Universal Robots PolyScope program: set_b_drawing_robot.urp

Program set_b_drawing_robot (installation=default directory=/programs createdIn=5.11.9.1010452 lastSavedIn=5.11.9.1010452 robotSerialNumber=20225200364)
Calibrated DH parameters: a=[0.00002, -0.569483, -0.54992, -0.00001, -0.000036, 0]; d=[0.180894, -146.691669, 192.918669, -46.053088, 0.119778, 0.115602]; alpha=[1.571425, -0.001534, 0.003359, 1.568739, -1.571477, 0]; deltaTheta=[0, 0.376258, -0.101074, -0.275185, -0.000002, 0]
Robot Program (runOnlyOnce=true)
  Script file /programs/set_b_drawing_robot.script_bak
    | def Machining3():
    |   # Default parameters:
    |   global speed_ms = 0.3
    |   global speed_rads = 0.75
    |   global accel_mss = 3
    |   global accel_radss = 1.2
    |   global blend_radius_m = 0.00001
    | 
    |   # Add subprograms here
    |   # Start of main program
    |   # Program generated by RoboDK v5.6.5 for UR10e on 17/10/2023 11:45:54
    |   # Using nominal kinematics.
    |   blend_radius_m = 0.001
    |   speed_ms = 1.000
    |   # set_reference(p[0.335000, -0.154000, -0.015000, 0.000000, 0.000000, 0.000000])
    |   set_tcp(p[0.000000, 0.000000, 0.252000, 0.000000, 0.000000, 0.000000])
    |   # Show Tool
    |   movej([0.061043, -1.072595, -2.581751, -1.058043, 1.570796, 1.631840],accel_radss,speed_rads,0,blend_radius_m)
    |   movel([0.061043, -1.163101, -2.647930, -0.901358, 1.570796, 1.631840],accel_mss,speed_ms,0,blend_radius_m)
    |   speed_ms = 1.000
    |   speed_ms = 0.005
    |   movel([0.061043, -1.123091, -2.622268, -0.967030, 1.570796, 1.631840],accel_mss,speed_ms,0,blend_radius_m)
    |   speed_ms = 1.000
    |   movel([0.061043, -1.163101, -2.647930, -0.901358, 1.570796, 1.631840],accel_mss,speed_ms,0,blend_radius_m)
    |   speed_ms = 0.040
    |   speed_ms = 1.000
    |   movel([0.083343, -1.403315, -2.504510, -0.804564, 1.570796, 1.654139],accel_mss,speed_ms,0,blend_radius_m)
    |   speed_ms = 0.005
    |   movel([0.083343, -1.443044, -2.523768, -0.745577, 1.570796, 1.654139],accel_mss,speed_ms,0,blend_radius_m)
    |   speed_ms = 0.035
    |   movel([0.081487, -1.443536, -2.523375, -0.745478, 1.570796, 1.652283],accel_mss,speed_ms,0,blend_radius_m)
    |   movel([0.082098, -1.437213, -2.528399, -0.746777, 1.570796, 1.652894],accel_mss,speed_ms,0,blend_radius_m)
    |   movel([0.082718, -1.430832, -2.533407, -0.748150, 1.570796, 1.653514],accel_mss,speed_ms,0,blend_radius_m)
    |   movel([0.084603, -1.430324, -2.533803, -0.748261, 1.570796, 1.655399],accel_mss,speed_ms,0,blend_radius_m)
    |   movel([0.086489, -1.429818, -2.534197, -0.748373, 1.570796, 1.657285],accel_mss,speed_ms,0,blend_radius_m)
    |   movel([0.085840, -1.436215, -2.529186, -0.746988, 1.570796, 1.656636],accel_mss,speed_ms,0,blend_radius_m)
    |   movel([0.085200, -1.442554, -2.524159, -0.745676, 1.570796, 1.655996],accel_mss,speed_ms,0,blend_radius_m)
    |   movel([0.083343, -1.443044, -2.523768, -0.745577, 1.570796, 1.654139],accel_mss,speed_ms,0,blend_radius_m)
    |   movel([0.081487, -1.443536, -2.523375, -0.745478, 1.570796, 1.652283],accel_mss,speed_ms,0,blend_radius_m)
    |   movel([0.081525, -1.443142, -2.523689, -0.745557, 1.570796, 1.652321],accel_mss,speed_ms,0,blend_radius_m)
    |   speed_ms = 0.005
    |   movel([0.081525, -1.434929, -2.519954, -0.757506, 1.570796, 1.652321],accel_mss,speed_ms,0,blend_radius_m)
    |   speed_ms = 0.040
    |   movel([0.115333, -1.443644, -2.513024, -0.755721, 1.570796, 1.686129],accel_mss,speed_ms,0,blend_radius_m)
    |   speed_ms = 0.005
    |   movel([0.115333, -1.451791, -2.516723, -0.743874, 1.570796, 1.686129],accel_mss,speed_ms,0,blend_radius_m)
    |   speed_ms = 0.035
    |   movel([0.102885, -1.454661, -2.514387, -0.743341, 1.570796, 1.673681],accel_mss,speed_ms,0,blend_radius_m)
    |   movel([0.102970, -1.452841, -2.515871, -0.743678, 1.570796, 1.673766],accel_mss,speed_ms,0,blend_radius_m)
    |   movel([0.103055, -1.451016, -2.517353, -0.744021, 1.570796, 1.673851],accel_mss,speed_ms,0,blend_radius_m)
    |   movel([0.115713, -1.447978, -2.519809, -0.744602, 1.570796, 1.686509],accel_mss,speed_ms,0,blend_radius_m)
    |   movel([0.128398, -1.445051, -2.522162, -0.745176, 1.570796, 1.699194],accel_mss,speed_ms,0,blend_radius_m)
    |   movel([0.128100, -1.447044, -2.520561, -0.744784, 1.570796, 1.698897],accel_mss,speed_ms,0,blend_radius_m)
    |   movel([0.127804, -1.449031, -2.518959, -0.744399, 1.570796, 1.698600],accel_mss,speed_ms,0,blend_radius_m)
    |   movel([0.115333, -1.451791, -2.516723, -0.743874, 1.570796, 1.686129],accel_mss,speed_ms,0,blend_radius_m)
    |   movel([0.113047, -1.452309, -2.516303, -0.743777, 1.570796, 1.683843],accel_mss,speed_ms,0,blend_radius_m)
    |   speed_ms = 0.005
    |   movel([0.113047, -1.444166, -2.512605, -0.755618, 1.570796, 1.683843],accel_mss,speed_ms,0,blend_radius_m)
    |   speed_ms = 0.040
    |   movel([0.116068, -1.438174, -2.517387, -0.756828, 1.570796, 1.686864],accel_mss,speed_ms,0,blend_radius_m)
    |   speed_ms = 0.005
    |   movel([0.116068, -1.446363, -2.521109, -0.744917, 1.570796, 1.686864],accel_mss,speed_ms,0,blend_radius_m)
    |   speed_ms = 0.035
    |   movel([0.086775, -1.453581, -2.515268, -0.743540, 1.570796, 1.657571],accel_mss,speed_ms,0,blend_radius_m)
    |   movel([0.089171, -1.430471, -2.533689, -0.748229, 1.570796, 1.659968],accel_mss,speed_ms,0,blend_radius_m)
    |   movel([0.091706, -1.406568, -2.551895, -0.753926, 1.570796, 1.662503],accel_mss,speed_ms,0,blend_radius_m)
    |   movel([0.122816, -1.398387, -2.557932, -0.756070, 1.570796, 1.693612],accel_mss,speed_ms,0,blend_radius_m)
    |   movel([0.154099, -1.390862, -2.563398, -0.758129, 1.570796, 1.724895],accel_mss,speed_ms,0,blend_radius_m)
    |   movel([0.149681, -1.415746, -2.545005, -0.751638, 1.570796, 1.720477],accel_mss,speed_ms,0,blend_radius_m)
    |   movel([0.145508, -1.439740, -2.526398, -0.746251, 1.570796, 1.716304],accel_mss,speed_ms,0,blend_radius_m)
    |   movel([0.116068, -1.446363, -2.521109, -0.744917, 1.570796, 1.686864],accel_mss,speed_ms,0,blend_radius_m)
    |   movel([0.113764, -1.446908, -2.520670, -0.744811, 1.570796, 1.684560],accel_mss,speed_ms,0,blend_radius_m)
    |   speed_ms = 0.005
    |   movel([0.113764, -1.438723, -2.516951, -0.756715, 1.570796, 1.684560],accel_mss,speed_ms,0,blend_radius_m)
    |   speed_ms = 0.040
    |   movel([0.108373, -1.429267, -2.524395, -0.758727, 1.570796, 1.679169],accel_mss,speed_ms,0,blend_radius_m)
    |   speed_ms = 0.005
    |   movel([0.108373, -1.437523, -2.528153, -0.746712, 1.570796, 1.679169],accel_mss,speed_ms,0,blend_radius_m)
    |   speed_ms = 0.035
    |   movel([0.107038, -1.438547, -2.527344, -0.746498, 1.570796, 1.677835],accel_mss,speed_ms,0,blend_radius_m)
    |   movel([0.106310, -1.438957, -2.527019, -0.746413, 1.570796, 1.677107],accel_mss,speed_ms,0,blend_radius_m)
    |   movel([0.104799, -1.439542, -2.526555, -0.746292, 1.570796, 1.675596],accel_mss,speed_ms,0,blend_radius_m)
    |   movel([0.104044, -1.439704, -2.526426, -0.746258, 1.570796, 1.674840],accel_mss,speed_ms,0,blend_radius_m)
    |   movel([0.102614, -1.439758, -2.526384, -0.746247, 1.570796, 1.673411],accel_mss,speed_ms,0,blend_radius_m)
    |   movel([0.101980, -1.439648, -2.526471, -0.746270, 1.570796, 1.672776],accel_mss,speed_ms,0,blend_radius_m)
    |   movel([0.100905, -1.439161, -2.526857, -0.746371, 1.570796, 1.671701],accel_mss,speed_ms,0,blend_radius_m)
    |   movel([0.100487, -1.438793, -2.527149, -0.746447, 1.570796, 1.671284],accel_mss,speed_ms,0,blend_radius_m)
    |   movel([0.099966, -1.437859, -2.527888, -0.746642, 1.570796, 1.670762],accel_mss,speed_ms,0,blend_radius_m)
    |   movel([0.099866, -1.437301, -2.528329, -0.746759, 1.570796, 1.670663],accel_mss,speed_ms,0,blend_radius_m)
    |   movel([0.099878, -1.436700, -2.528804, -0.746885, 1.570796, 1.670674],accel_mss,speed_ms,0,blend_radius_m)
    |   movel([0.100054, -1.435839, -2.529482, -0.747068, 1.570796, 1.670850],accel_mss,speed_ms,0,blend_radius_m)
    |   movel([0.100376, -1.435105, -2.530060, -0.747224, 1.570796, 1.671172],accel_mss,speed_ms,0,blend_radius_m)
    |   movel([0.100937, -1.434333, -2.530667, -0.747389, 1.570796, 1.671733],accel_mss,speed_ms,0,blend_radius_m)
    |   movel([0.101867, -1.433331, -2.531453, -0.747605, 1.570796, 1.672664],accel_mss,speed_ms,0,blend_radius_m)
    |   movel([0.103005, -1.432248, -2.532301, -0.747840, 1.570796, 1.673801],accel_mss,speed_ms,0,blend_radius_m)
    |   movel([0.103766, -1.431710, -2.532722, -0.747957, 1.570796, 1.674563],accel_mss,speed_ms,0,blend_radius_m)
    |   movel([0.104600, -1.431387, -2.532974, -0.748028, 1.570796, 1.675397],accel_mss,speed_ms,0,blend_radius_m)
    |   movel([0.106011, -1.431098, -2.533199, -0.748091, 1.570796, 1.676807],accel_mss,speed_ms,0,blend_radius_m)
    |   movel([0.107167, -1.430973, -2.533297, -0.748119, 1.570796, 1.677964],accel_mss,speed_ms,0,blend_radius_m)
    |   movel([0.108266, -1.430998, -2.533278, -0.748113, 1.570796, 1.679062],accel_mss,speed_ms,0,blend_radius_m)
    |   movel([0.109099, -1.431186, -2.533131, -0.748072, 1.570796, 1.679896],accel_mss,speed_ms,0,blend_radius_m)
    |   movel([0.109775, -1.431571, -2.532831, -0.747988, 1.570796, 1.680572],accel_mss,speed_ms,0,blend_radius_m)
    |   movel([0.110228, -1.432115, -2.532405, -0.747869, 1.570796, 1.681024],accel_mss,speed_ms,0,blend_radius_m)
    |   movel([0.110459, -1.432805, -2.531865, -0.747719, 1.570796, 1.681255],accel_mss,speed_ms,0,blend_radius_m)
    |   movel([0.110489, -1.433683, -2.531177, -0.747529, 1.570796, 1.681285],accel_mss,speed_ms,0,blend_radius_m)
    |   movel([0.110328, -1.434616, -2.530445, -0.747328, 1.570796, 1.681124],accel_mss,speed_ms,0,blend_radius_m)
    |   movel([0.110059, -1.435334, -2.529880, -0.747175, 1.570796, 1.680855],accel_mss,speed_ms,0,blend_radius_m)
    |   movel([0.109634, -1.436071, -2.529299, -0.747018, 1.570796, 1.680430],accel_mss,speed_ms,0,blend_radius_m)
    |   movel([0.109064, -1.436811, -2.528716, -0.746862, 1.570796, 1.679861],accel_mss,speed_ms,0,blend_radius_m)
    |   movel([0.108373, -1.437523, -2.528153, -0.746712, 1.570796, 1.679169],accel_mss,speed_ms,0,blend_radius_m)
    |   movel([0.107038, -1.438547, -2.527344, -0.746498, 1.570796, 1.677835],accel_mss,speed_ms,0,blend_radius_m)
    |   movel([0.106310, -1.438957, -2.527019, -0.746413, 1.570796, 1.677107],accel_mss,speed_ms,0,blend_radius_m)
    |   speed_ms = 0.005
    |   movel([0.106310, -1.430712, -2.523266, -0.758411, 1.570796, 1.677107],accel_mss,speed_ms,0,blend_radius_m)
    |   speed_ms = 0.040
    |   movel([0.108450, -1.424967, -2.527736, -0.759686, 1.570796, 1.679246],accel_mss,speed_ms,0,blend_radius_m)
    |   speed_ms = 0.005
    |   movel([0.108450, -1.433255, -2.531513, -0.747621, 1.570796, 1.679246],accel_mss,speed_ms,0,blend_radius_m)
    |   speed_ms = 0.035
    |   movel([0.108678, -1.434176, -2.530790, -0.747423, 1.570796, 1.679474],accel_mss,speed_ms,0,blend_radius_m)
    |   movel([0.108589, -1.434982, -2.530157, -0.747250, 1.570796, 1.679385],accel_mss,speed_ms,0,blend_radius_m)
    |   movel([0.108163, -1.435793, -2.529519, -0.747077, 1.570796, 1.678959],accel_mss,speed_ms,0,blend_radius_m)
    |   movel([0.107355, -1.436726, -2.528783, -0.746880, 1.570796, 1.678151],accel_mss,speed_ms,0,blend_radius_m)
    |   movel([0.106463, -1.437462, -2.528202, -0.746725, 1.570796, 1.677259],accel_mss,speed_ms,0,blend_radius_m)
    |   movel([0.105461, -1.438014, -2.527765, -0.746609, 1.570796, 1.676258],accel_mss,speed_ms,0,blend_radius_m)
    |   movel([0.104454, -1.438323, -2.527521, -0.746545, 1.570796, 1.675251],accel_mss,speed_ms,0,blend_radius_m)
    |   movel([0.103505, -1.438364, -2.527489, -0.746536, 1.570796, 1.674302],accel_mss,speed_ms,0,blend_radius_m)
    |   movel([0.102703, -1.438137, -2.527668, -0.746584, 1.570796, 1.673500],accel_mss,speed_ms,0,blend_radius_m)
    |   movel([0.102119, -1.437659, -2.528047, -0.746684, 1.570796, 1.672915],accel_mss,speed_ms,0,blend_radius_m)
    |   movel([0.101790, -1.436965, -2.528595, -0.746830, 1.570796, 1.672586],accel_mss,speed_ms,0,blend_radius_m)
    |   movel([0.101749, -1.436130, -2.529253, -0.747006, 1.570796, 1.672545],accel_mss,speed_ms,0,blend_radius_m)
    |   movel([0.101858, -1.435631, -2.529646, -0.747112, 1.570796, 1.672655],accel_mss,speed_ms,0,blend_radius_m)
    |   movel([0.102363, -1.434622, -2.530440, -0.747327, 1.570796, 1.673159],accel_mss,speed_ms,0,blend_radius_m)
    |   movel([0.102745, -1.434142, -2.530817, -0.747430, 1.570796, 1.673541],accel_mss,speed_ms,0,blend_radius_m)
    |   movel([0.103728, -1.433264, -2.531506, -0.747619, 1.570796, 1.674524],accel_mss,speed_ms,0,blend_radius_m)
    |   movel([0.104871, -1.432616, -2.532013, -0.747760, 1.570796, 1.675667],accel_mss,speed_ms,0,blend_radius_m)
    |   movel([0.106038, -1.432273, -2.532282, -0.747834, 1.570796, 1.676835],accel_mss,speed_ms,0,blend_radius_m)
    |   movel([0.107121, -1.432265, -2.532288, -0.747836, 1.570796, 1.677918],accel_mss,speed_ms,0,blend_radius_m)
    |   movel([0.107572, -1.432389, -2.532191, -0.747809, 1.570796, 1.678368],accel_mss,speed_ms,0,blend_radius_m)
    |   movel([0.107952, -1.432601, -2.532025, -0.747763, 1.570796, 1.678748],accel_mss,speed_ms,0,blend_radius_m)
    |   movel([0.108450, -1.433255, -2.531513, -0.747621, 1.570796, 1.679246],accel_mss,speed_ms,0,blend_radius_m)
    |   movel([0.108678, -1.434176, -2.530790, -0.747423, 1.570796, 1.679474],accel_mss,speed_ms,0,blend_radius_m)
    |   movel([0.108589, -1.434982, -2.530157, -0.747250, 1.570796, 1.679385],accel_mss,speed_ms,0,blend_radius_m)
    |   speed_ms = 0.005
    |   movel([0.108509, -1.426858, -2.526270, -0.759261, 1.570796, 1.679305],accel_mss,speed_ms,0,blend_radius_m)
    |   speed_ms = 0.040
    |   movel([0.111498, -1.422635, -2.529536, -0.760218, 1.570796, 1.682294],accel_mss,speed_ms,0,blend_radius_m)
    |   speed_ms = 0.005
    |   movel([0.111498, -1.430940, -2.533323, -0.748126, 1.570796, 1.682294],accel_mss,speed_ms,0,blend_radius_m)
    |   speed_ms = 0.035
    |   movel([0.111769, -1.431458, -2.532919, -0.748012, 1.570796, 1.682566],accel_mss,speed_ms,0,blend_radius_m)
    |   movel([0.112066, -1.432871, -2.531814, -0.747704, 1.570796, 1.682862],accel_mss,speed_ms,0,blend_radius_m)
    |   movel([0.112043, -1.433534, -2.531294, -0.747561, 1.570796, 1.682839],accel_mss,speed_ms,0,blend_radius_m)
    |   movel([0.111849, -1.434440, -2.530583, -0.747366, 1.570796, 1.682646],accel_mss,speed_ms,0,blend_radius_m)
    |   movel([0.111503, -1.435363, -2.529857, -0.747169, 1.570796, 1.682299],accel_mss,speed_ms,0,blend_radius_m)
    |   movel([0.111013, -1.436281, -2.529134, -0.746974, 1.570796, 1.681809],accel_mss,speed_ms,0,blend_radius_m)
    |   movel([0.110389, -1.437172, -2.528431, -0.746786, 1.570796, 1.681185],accel_mss,speed_ms,0,blend_radius_m)
    |   movel([0.109649, -1.438014, -2.527766, -0.746609, 1.570796, 1.680445],accel_mss,speed_ms,0,blend_radius_m)
    |   movel([0.108810, -1.438786, -2.527154, -0.746448, 1.570796, 1.679607],accel_mss,speed_ms,0,blend_radius_m)
    |   movel([0.107889, -1.439477, -2.526607, -0.746305, 1.570796, 1.678685],accel_mss,speed_ms,0,blend_radius_m)
    |   movel([0.106909, -1.440063, -2.526142, -0.746184, 1.570796, 1.677706],accel_mss,speed_ms,0,blend_radius_m)
    |   movel([0.105881, -1.440544, -2.525759, -0.746085, 1.570796, 1.676677],accel_mss,speed_ms,0,blend_radius_m)
    |   movel([0.104840, -1.440900, -2.525477, -0.746013, 1.570796, 1.675636],accel_mss,speed_ms,0,blend_radius_m)
    |   movel([0.103811, -1.441122, -2.525300, -0.745967, 1.570796, 1.674607],accel_mss,speed_ms,0,blend_radius_m)
    |   movel([0.102814, -1.441208, -2.525231, -0.745949, 1.570796, 1.673610],accel_mss,speed_ms,0,blend_radius_m)
    |   movel([0.101860, -1.441159, -2.525270, -0.745960, 1.570796, 1.672657],accel_mss,speed_ms,0,blend_radius_m)
    |   movel([0.100981, -1.440972, -2.525419, -0.745998, 1.570796, 1.671777],accel_mss,speed_ms,0,blend_radius_m)
    |   movel([0.100198, -1.440656, -2.525670, -0.746062, 1.570796, 1.670994],accel_mss,speed_ms,0,blend_radius_m)
    |   movel([0.099523, -1.440217, -2.526019, -0.746153, 1.570796, 1.670319],accel_mss,speed_ms,0,blend_radius_m)
    |   movel([0.098634, -1.439242, -2.526793, -0.746354, 1.570796, 1.669430],accel_mss,speed_ms,0,blend_radius_m)
    |   movel([0.098355, -1.438715, -2.527210, -0.746463, 1.570796, 1.669152],accel_mss,speed_ms,0,blend_radius_m)
    |   movel([0.098129, -1.437516, -2.528159, -0.746714, 1.570796, 1.668926],accel_mss,speed_ms,0,blend_radius_m)
    |   movel([0.098186, -1.436868, -2.528671, -0.746850, 1.570796, 1.668982],accel_mss,speed_ms,0,blend_radius_m)
    |   movel([0.098626, -1.435475, -2.529769, -0.747145, 1.570796, 1.669422],accel_mss,speed_ms,0,blend_radius_m)
    |   movel([0.099087, -1.434613, -2.530447, -0.747329, 1.570796, 1.669883],accel_mss,speed_ms,0,blend_radius_m)
    |   movel([0.099671, -1.433774, -2.531106, -0.747509, 1.570796, 1.670467],accel_mss,speed_ms,0,blend_radius_m)
    |   movel([0.100365, -1.432978, -2.531730, -0.747681, 1.570796, 1.671161],accel_mss,speed_ms,0,blend_radius_m)
    |   movel([0.101155, -1.432239, -2.532308, -0.747842, 1.570796, 1.671952],accel_mss,speed_ms,0,blend_radius_m)
    |   movel([0.102056, -1.431544, -2.532851, -0.747993, 1.570796, 1.672852],accel_mss,speed_ms,0,blend_radius_m)
    |   movel([0.103011, -1.430931, -2.533330, -0.748128, 1.570796, 1.673808],accel_mss,speed_ms,0,blend_radius_m)
    |   movel([0.104006, -1.430413, -2.533734, -0.748242, 1.570796, 1.674803],accel_mss,speed_ms,0,blend_radius_m)
    |   movel([0.105024, -1.429996, -2.534059, -0.748334, 1.570796, 1.675820],accel_mss,speed_ms,0,blend_radius_m)
    |   movel([0.106037, -1.429694, -2.534295, -0.748401, 1.570796, 1.676834],accel_mss,speed_ms,0,blend_radius_m)
    |   movel([0.107034, -1.429510, -2.534437, -0.748442, 1.570796, 1.677830],accel_mss,speed_ms,0,blend_radius_m)
    |   movel([0.108000, -1.429444, -2.534488, -0.748456, 1.570796, 1.678796],accel_mss,speed_ms,0,blend_radius_m)
    |   movel([0.108911, -1.429501, -2.534444, -0.748444, 1.570796, 1.679707],accel_mss,speed_ms,0,blend_radius_m)
    |   movel([0.109713, -1.429677, -2.534307, -0.748404, 1.570796, 1.680510],accel_mss,speed_ms,0,blend_radius_m)
    |   movel([0.110423, -1.429981, -2.534071, -0.748337, 1.570796, 1.681220],accel_mss,speed_ms,0,blend_radius_m)
    |   movel([0.111022, -1.430406, -2.533739, -0.748243, 1.570796, 1.681818],accel_mss,speed_ms,0,blend_radius_m)
    |   movel([0.111498, -1.430940, -2.533323, -0.748126, 1.570796, 1.682294],accel_mss,speed_ms,0,blend_radius_m)
    |   movel([0.111769, -1.431458, -2.532919, -0.748012, 1.570796, 1.682566],accel_mss,speed_ms,0,blend_radius_m)
    |   movel([0.112020, -1.432648, -2.531988, -0.747753, 1.570796, 1.682816],accel_mss,speed_ms,0,blend_radius_m)
    |   speed_ms = 0.005
    |   movel([0.112020, -1.424355, -2.528209, -0.759825, 1.570796, 1.682816],accel_mss,speed_ms,0,blend_radius_m)
    |   speed_ms = 0.040
    |   movel([0.118670, -1.415194, -2.535227, -0.761968, 1.570796, 1.689466],accel_mss,speed_ms,0,blend_radius_m)
    |   speed_ms = 0.005
    |   movel([0.118670, -1.423554, -2.539045, -0.749790, 1.570796, 1.689466],accel_mss,speed_ms,0,blend_radius_m)
    |   speed_ms = 0.035
    |   movel([0.124083, -1.422246, -2.540050, -0.750093, 1.570796, 1.694879],accel_mss,speed_ms,0,blend_radius_m)
    |   movel([0.117797, -1.433318, -2.531463, -0.747608, 1.570796, 1.688593],accel_mss,speed_ms,0,blend_radius_m)
    |   movel([0.117485, -1.433740, -2.531132, -0.747517, 1.570796, 1.688282],accel_mss,speed_ms,0,blend_radius_m)
    |   movel([0.116691, -1.432642, -2.531993, -0.747754, 1.570796, 1.687488],accel_mss,speed_ms,0,blend_radius_m)
    |   movel([0.115225, -1.429498, -2.534447, -0.748444, 1.570796, 1.686021],accel_mss,speed_ms,0,blend_radius_m)
    |   movel([0.113262, -1.424883, -2.538022, -0.749484, 1.570796, 1.684058],accel_mss,speed_ms,0,blend_radius_m)
    |   movel([0.118670, -1.423554, -2.539045, -0.749790, 1.570796, 1.689466],accel_mss,speed_ms,0,blend_radius_m)
    |   movel([0.121038, -1.422979, -2.539487, -0.749923, 1.570796, 1.691834],accel_mss,speed_ms,0,blend_radius_m)
    |   speed_ms = 0.005
    |   movel([0.121038, -1.414614, -2.535667, -0.762108, 1.570796, 1.691834],accel_mss,speed_ms,0,blend_radius_m)
    |   speed_ms = 0.040
    |   movel([0.134556, -1.418951, -2.532364, -0.761074, 1.570796, 1.705352],accel_mss,speed_ms,0,blend_radius_m)
    |   speed_ms = 0.005
    |   movel([0.134556, -1.427284, -2.536166, -0.748939, 1.570796, 1.705352],accel_mss,speed_ms,0,blend_radius_m)
    |   speed_ms = 0.035
    |   movel([0.134713, -1.428009, -2.535604, -0.748776, 1.570796, 1.705509],accel_mss,speed_ms,0,blend_radius_m)
    |   movel([0.134561, -1.428836, -2.534961, -0.748591, 1.570796, 1.705357],accel_mss,speed_ms,0,blend_radius_m)
    |   movel([0.134112, -1.429713, -2.534279, -0.748397, 1.570796, 1.704908],accel_mss,speed_ms,0,blend_radius_m)
    |   movel([0.133429, -1.430532, -2.533641, -0.748216, 1.570796, 1.704225],accel_mss,speed_ms,0,blend_radius_m)
    |   movel([0.132541, -1.431249, -2.533082, -0.748058, 1.570796, 1.703337],accel_mss,speed_ms,0,blend_radius_m)
    |   movel([0.131550, -1.431787, -2.532662, -0.747940, 1.570796, 1.702346],accel_mss,speed_ms,0,blend_radius_m)
    |   movel([0.130539, -1.432096, -2.532420, -0.747873, 1.570796, 1.701335],accel_mss,speed_ms,0,blend_radius_m)
    |   movel([0.129581, -1.432154, -2.532375, -0.747860, 1.570796, 1.700377],accel_mss,speed_ms,0,blend_radius_m)
    |   movel([0.128793, -1.431956, -2.532529, -0.747903, 1.570796, 1.699589],accel_mss,speed_ms,0,blend_radius_m)
    |   movel([0.128207, -1.431521, -2.532870, -0.747999, 1.570796, 1.699003],accel_mss,speed_ms,0,blend_radius_m)
    |   movel([0.127885, -1.430887, -2.533365, -0.748138, 1.570796, 1.698681],accel_mss,speed_ms,0,blend_radius_m)
    |   movel([0.127854, -1.430106, -2.533974, -0.748310, 1.570796, 1.698650],accel_mss,speed_ms,0,blend_radius_m)
    |   movel([0.128121, -1.429207, -2.534673, -0.748509, 1.570796, 1.698917],accel_mss,speed_ms,0,blend_radius_m)
    |   movel([0.128656, -1.428312, -2.535368, -0.748708, 1.570796, 1.699452],accel_mss,speed_ms,0,blend_radius_m)
    |   movel([0.129437, -1.427445, -2.536041, -0.748903, 1.570796, 1.700234],accel_mss,speed_ms,0,blend_radius_m)
    |   movel([0.130376, -1.426701, -2.536617, -0.749071, 1.570796, 1.701173],accel_mss,speed_ms,0,blend_radius_m)
    |   movel([0.131197, -1.426193, -2.537010, -0.749186, 1.570796, 1.701993],accel_mss,speed_ms,0,blend_radius_m)
    |   movel([0.131729, -1.425980, -2.537174, -0.749234, 1.570796, 1.702526],accel_mss,speed_ms,0,blend_radius_m)
    |   movel([0.132234, -1.425952, -2.537196, -0.749240, 1.570796, 1.703030],accel_mss,speed_ms,0,blend_radius_m)
    |   movel([0.133441, -1.426292, -2.536934, -0.749163, 1.570796, 1.704237],accel_mss,speed_ms,0,blend_radius_m)
    |   movel([0.133917, -1.426587, -2.536706, -0.749097, 1.570796, 1.704714],accel_mss,speed_ms,0,blend_radius_m)
    |   movel([0.134556, -1.427284, -2.536166, -0.748939, 1.570796, 1.705352],accel_mss,speed_ms,0,blend_radius_m)
    |   movel([0.134713, -1.428009, -2.535604, -0.748776, 1.570796, 1.705509],accel_mss,speed_ms,0,blend_radius_m)
    |   movel([0.134561, -1.428836, -2.534961, -0.748591, 1.570796, 1.705357],accel_mss,speed_ms,0,blend_radius_m)
    |   movel([0.134352, -1.429244, -2.534645, -0.748501, 1.570796, 1.705149],accel_mss,speed_ms,0,blend_radius_m)
    |   speed_ms = 0.005
    |   movel([0.134352, -1.420925, -2.530851, -0.760613, 1.570796, 1.705149],accel_mss,speed_ms,0,blend_radius_m)
    |   speed_ms = 0.040
    |   movel([0.135995, -1.421177, -2.530658, -0.760554, 1.570796, 1.706791],accel_mss,speed_ms,0,blend_radius_m)
    |   speed_ms = 0.005
    |   movel([0.135995, -1.429493, -2.534450, -0.748445, 1.570796, 1.706791],accel_mss,speed_ms,0,blend_radius_m)
    |   speed_ms = 0.035
    |   movel([0.136640, -1.428314, -2.535367, -0.748708, 1.570796, 1.707437],accel_mss,speed_ms,0,blend_radius_m)
    |   movel([0.136842, -1.427711, -2.535835, -0.748843, 1.570796, 1.707638],accel_mss,speed_ms,0,blend_radius_m)
    |   movel([0.136811, -1.427161, -2.536261, -0.748967, 1.570796, 1.707608],accel_mss,speed_ms,0,blend_radius_m)
    |   movel([0.136224, -1.425707, -2.537385, -0.749296, 1.570796, 1.707020],accel_mss,speed_ms,0,blend_radius_m)
    |   movel([0.135852, -1.425300, -2.537700, -0.749389, 1.570796, 1.706648],accel_mss,speed_ms,0,blend_radius_m)
    |   movel([0.135381, -1.424981, -2.537946, -0.749462, 1.570796, 1.706178],accel_mss,speed_ms,0,blend_radius_m)
    |   movel([0.134822, -1.424761, -2.538115, -0.749512, 1.570796, 1.705618],accel_mss,speed_ms,0,blend_radius_m)
    |   movel([0.133426, -1.424588, -2.538249, -0.749552, 1.570796, 1.704223],accel_mss,speed_ms,0,blend_radius_m)
    |   movel([0.132662, -1.424644, -2.538206, -0.749539, 1.570796, 1.703458],accel_mss,speed_ms,0,blend_radius_m)
    |   movel([0.131068, -1.425036, -2.537904, -0.749449, 1.570796, 1.701864],accel_mss,speed_ms,0,blend_radius_m)
    |   movel([0.130262, -1.425364, -2.537651, -0.749374, 1.570796, 1.701059],accel_mss,speed_ms,0,blend_radius_m)
    |   movel([0.128715, -1.426256, -2.536961, -0.749172, 1.570796, 1.699511],accel_mss,speed_ms,0,blend_radius_m)
    |   movel([0.128048, -1.426777, -2.536558, -0.749054, 1.570796, 1.698845],accel_mss,speed_ms,0,blend_radius_m)
    |   movel([0.127449, -1.427357, -2.536109, -0.748923, 1.570796, 1.698245],accel_mss,speed_ms,0,blend_radius_m)
    |   movel([0.126929, -1.427983, -2.535624, -0.748782, 1.570796, 1.697725],accel_mss,speed_ms,0,blend_radius_m)
    |   movel([0.126501, -1.428638, -2.535116, -0.748636, 1.570796, 1.697298],accel_mss,speed_ms,0,blend_radius_m)
    |   movel([0.126013, -1.429754, -2.534248, -0.748388, 1.570796, 1.696809],accel_mss,speed_ms,0,blend_radius_m)
    |   movel([0.125816, -1.430837, -2.533404, -0.748149, 1.570796, 1.696612],accel_mss,speed_ms,0,blend_radius_m)
    |   movel([0.125934, -1.431780, -2.532667, -0.747942, 1.570796, 1.696730],accel_mss,speed_ms,0,blend_radius_m)
    |   movel([0.126370, -1.432553, -2.532063, -0.747774, 1.570796, 1.697166],accel_mss,speed_ms,0,blend_radius_m)
    |   movel([0.127106, -1.433124, -2.531616, -0.747650, 1.570796, 1.697902],accel_mss,speed_ms,0,blend_radius_m)
    |   movel([0.128073, -1.433435, -2.531372, -0.747582, 1.570796, 1.698870],accel_mss,speed_ms,0,blend_radius_m)
    |   movel([0.129278, -1.433498, -2.531322, -0.747569, 1.570796, 1.700074],accel_mss,speed_ms,0,blend_radius_m)
    |   movel([0.130573, -1.433316, -2.531465, -0.747608, 1.570796, 1.701369],accel_mss,speed_ms,0,blend_radius_m)
    |   movel([0.132350, -1.432755, -2.531905, -0.747730, 1.570796, 1.703146],accel_mss,speed_ms,0,blend_radius_m)
    |   movel([0.133094, -1.432405, -2.532178, -0.747806, 1.570796, 1.703890],accel_mss,speed_ms,0,blend_radius_m)
    |   movel([0.133806, -1.431961, -2.532525, -0.747902, 1.570796, 1.704602],accel_mss,speed_ms,0,blend_radius_m)
    |   movel([0.134437, -1.431458, -2.532919, -0.748012, 1.570796, 1.705233],accel_mss,speed_ms,0,blend_radius_m)
    |   movel([0.134998, -1.430887, -2.533364, -0.748137, 1.570796, 1.705795],accel_mss,speed_ms,0,blend_radius_m)
    |   movel([0.135995, -1.429493, -2.534450, -0.748445, 1.570796, 1.706791],accel_mss,speed_ms,0,blend_radius_m)
    |   movel([0.136640, -1.428314, -2.535367, -0.748708, 1.570796, 1.707437],accel_mss,speed_ms,0,blend_radius_m)
    |   movel([0.136842, -1.427711, -2.535835, -0.748843, 1.570796, 1.707638],accel_mss,speed_ms,0,blend_radius_m)
    |   movel([0.136827, -1.427423, -2.536058, -0.748908, 1.570796, 1.707623],accel_mss,speed_ms,0,blend_radius_m)
    |   speed_ms = 0.005
    |   movel([0.136827, -1.419092, -2.532256, -0.761041, 1.570796, 1.707623],accel_mss,speed_ms,0,blend_radius_m)
    |   speed_ms = 0.040
    |   movel([0.151093, -1.418454, -2.532744, -0.761191, 1.570796, 1.721889],accel_mss,speed_ms,0,blend_radius_m)
    |   speed_ms = 0.005
    |   movel([0.151093, -1.426790, -2.536548, -0.749051, 1.570796, 1.721889],accel_mss,speed_ms,0,blend_radius_m)
    |   speed_ms = 0.035
    |   movel([0.149215, -1.427195, -2.536234, -0.748959, 1.570796, 1.720011],accel_mss,speed_ms,0,blend_radius_m)
    |   movel([0.150353, -1.420598, -2.541312, -0.750479, 1.570796, 1.721149],accel_mss,speed_ms,0,blend_radius_m)
    |   movel([0.151509, -1.413936, -2.546374, -0.752079, 1.570796, 1.722305],accel_mss,speed_ms,0,blend_radius_m)
    |   movel([0.153417, -1.413517, -2.546690, -0.752182, 1.570796, 1.724214],accel_mss,speed_ms,0,blend_radius_m)
    |   movel([0.155326, -1.413100, -2.547004, -0.752285, 1.570796, 1.726122],accel_mss,speed_ms,0,blend_radius_m)
    |   movel([0.154140, -1.419776, -2.541940, -0.750672, 1.570796, 1.724936],accel_mss,speed_ms,0,blend_radius_m)
    |   movel([0.152972, -1.426387, -2.536860, -0.749142, 1.570796, 1.723768],accel_mss,speed_ms,0,blend_radius_m)
    |   movel([0.151093, -1.426790, -2.536548, -0.749051, 1.570796, 1.721889],accel_mss,speed_ms,0,blend_radius_m)
    |   movel([0.149215, -1.427195, -2.536234, -0.748959, 1.570796, 1.720011],accel_mss,speed_ms,0,blend_radius_m)
    |   movel([0.149285, -1.426785, -2.536552, -0.749052, 1.570796, 1.720082],accel_mss,speed_ms,0,blend_radius_m)
    |   speed_ms = 0.005
    |   movel([0.149285, -1.418448, -2.532748, -0.761192, 1.570796, 1.720082],accel_mss,speed_ms,0,blend_radius_m)
    |   speed_ms = 0.040
    |   movel([0.138194, -1.417141, -2.533746, -0.761502, 1.570796, 1.708991],accel_mss,speed_ms,0,blend_radius_m)
    |   speed_ms = 0.005
    |   movel([0.138194, -1.425487, -2.537556, -0.749346, 1.570796, 1.708991],accel_mss,speed_ms,0,blend_radius_m)
    |   speed_ms = 0.035
    |   movel([0.137776, -1.424690, -2.538171, -0.749529, 1.570796, 1.708572],accel_mss,speed_ms,0,blend_radius_m)
    |   movel([0.137130, -1.424063, -2.538653, -0.749672, 1.570796, 1.707926],accel_mss,speed_ms,0,blend_radius_m)
    |   movel([0.136238, -1.423570, -2.539033, -0.749786, 1.570796, 1.707034],accel_mss,speed_ms,0,blend_radius_m)
    |   movel([0.135198, -1.423260, -2.539272, -0.749858, 1.570796, 1.705994],accel_mss,speed_ms,0,blend_radius_m)
    |   movel([0.134027, -1.423137, -2.539366, -0.749886, 1.570796, 1.704823],accel_mss,speed_ms,0,blend_radius_m)
    |   movel([0.132767, -1.423207, -2.539312, -0.749870, 1.570796, 1.703563],accel_mss,speed_ms,0,blend_radius_m)
    |   movel([0.131525, -1.423470, -2.539110, -0.749809, 1.570796, 1.702321],accel_mss,speed_ms,0,blend_radius_m)
    |   movel([0.130268, -1.423937, -2.538750, -0.749701, 1.570796, 1.701064],accel_mss,speed_ms,0,blend_radius_m)
    |   movel([0.129210, -1.424482, -2.538331, -0.749576, 1.570796, 1.700007],accel_mss,speed_ms,0,blend_radius_m)
    |   movel([0.128199, -1.425138, -2.537825, -0.749426, 1.570796, 1.698995],accel_mss,speed_ms,0,blend_radius_m)
    |   movel([0.127256, -1.425893, -2.537242, -0.749254, 1.570796, 1.698052],accel_mss,speed_ms,0,blend_radius_m)
    |   movel([0.126405, -1.426724, -2.536599, -0.749066, 1.570796, 1.697201],accel_mss,speed_ms,0,blend_radius_m)
    |   movel([0.125686, -1.427595, -2.535925, -0.748869, 1.570796, 1.696483],accel_mss,speed_ms,0,blend_radius_m)
    |   movel([0.125101, -1.428505, -2.535218, -0.748665, 1.570796, 1.695898],accel_mss,speed_ms,0,blend_radius_m)
    |   movel([0.124667, -1.429433, -2.534497, -0.748459, 1.570796, 1.695464],accel_mss,speed_ms,0,blend_radius_m)
    |   movel([0.124391, -1.430353, -2.533781, -0.748255, 1.570796, 1.695187],accel_mss,speed_ms,0,blend_radius_m)
    |   movel([0.124284, -1.431236, -2.533092, -0.748061, 1.570796, 1.695080],accel_mss,speed_ms,0,blend_radius_m)
    |   movel([0.124345, -1.432063, -2.532446, -0.747880, 1.570796, 1.695142],accel_mss,speed_ms,0,blend_radius_m)
    |   movel([0.124576, -1.432812, -2.531860, -0.747717, 1.570796, 1.695372],accel_mss,speed_ms,0,blend_radius_m)
    |   movel([0.124968, -1.433462, -2.531350, -0.747576, 1.570796, 1.695764],accel_mss,speed_ms,0,blend_radius_m)
    |   movel([0.125516, -1.434019, -2.530914, -0.747457, 1.570796, 1.696313],accel_mss,speed_ms,0,blend_radius_m)
    |   movel([0.126197, -1.434455, -2.530571, -0.747363, 1.570796, 1.696993],accel_mss,speed_ms,0,blend_radius_m)
    |   movel([0.126988, -1.434761, -2.530331, -0.747297, 1.570796, 1.697785],accel_mss,speed_ms,0,blend_radius_m)
    |   movel([0.127878, -1.434927, -2.530200, -0.747262, 1.570796, 1.698675],accel_mss,speed_ms,0,blend_radius_m)
    |   movel([0.128797, -1.434959, -2.530175, -0.747255, 1.570796, 1.699593],accel_mss,speed_ms,0,blend_radius_m)
    |   movel([0.129766, -1.434867, -2.530247, -0.747275, 1.570796, 1.700562],accel_mss,speed_ms,0,blend_radius_m)
    |   movel([0.130764, -1.434656, -2.530413, -0.747320, 1.570796, 1.701560],accel_mss,speed_ms,0,blend_radius_m)
    |   movel([0.131774, -1.434324, -2.530674, -0.747391, 1.570796, 1.702570],accel_mss,speed_ms,0,blend_radius_m)
    |   movel([0.132774, -1.433883, -2.531020, -0.747486, 1.570796, 1.703570],accel_mss,speed_ms,0,blend_radius_m)
    |   movel([0.133750, -1.433337, -2.531448, -0.747603, 1.570796, 1.704546],accel_mss,speed_ms,0,blend_radius_m)
    |   movel([0.134679, -1.432699, -2.531948, -0.747742, 1.570796, 1.705475],accel_mss,speed_ms,0,blend_radius_m)
    |   movel([0.135547, -1.431980, -2.532511, -0.747898, 1.570796, 1.706343],accel_mss,speed_ms,0,blend_radius_m)
    |   movel([0.136306, -1.431215, -2.533108, -0.748065, 1.570796, 1.707102],accel_mss,speed_ms,0,blend_radius_m)
    |   movel([0.136968, -1.430399, -2.533745, -0.748245, 1.570796, 1.707765],accel_mss,speed_ms,0,blend_radius_m)
    |   movel([0.137520, -1.429546, -2.534410, -0.748434, 1.570796, 1.708316],accel_mss,speed_ms,0,blend_radius_m)
    |   movel([0.137950, -1.428674, -2.535087, -0.748628, 1.570796, 1.708747],accel_mss,speed_ms,0,blend_radius_m)
    |   movel([0.138233, -1.427824, -2.535747, -0.748818, 1.570796, 1.709030],accel_mss,speed_ms,0,blend_radius_m)
    |   movel([0.138370, -1.426997, -2.536388, -0.749004, 1.570796, 1.709167],accel_mss,speed_ms,0,blend_radius_m)
    |   movel([0.138358, -1.426210, -2.536997, -0.749182, 1.570796, 1.709154],accel_mss,speed_ms,0,blend_radius_m)
    |   movel([0.138194, -1.425487, -2.537556, -0.749346, 1.570796, 1.708991],accel_mss,speed_ms,0,blend_radius_m)
    |   movel([0.137776, -1.424690, -2.538171, -0.749529, 1.570796, 1.708572],accel_mss,speed_ms,0,blend_radius_m)
    |   movel([0.137158, -1.424088, -2.538634, -0.749667, 1.570796, 1.707954],accel_mss,speed_ms,0,blend_radius_m)
    |   speed_ms = 0.005
    |   movel([0.137158, -1.415732, -2.534818, -0.761839, 1.570796, 1.707954],accel_mss,speed_ms,0,blend_radius_m)
    |   speed_ms = 0.040
    |   movel([0.135389, -1.401511, -2.545479, -0.765399, 1.570796, 1.706186],accel_mss,speed_ms,0,blend_radius_m)
    |   speed_ms = 0.005
    |   movel([0.135389, -1.409972, -2.549355, -0.753063, 1.570796, 1.706186],accel_mss,speed_ms,0,blend_radius_m)
    |   speed_ms = 0.035
    |   movel([0.135900, -1.410093, -2.549263, -0.753032, 1.570796, 1.706696],accel_mss,speed_ms,0,blend_radius_m)
    |   movel([0.136203, -1.410331, -2.549085, -0.752973, 1.570796, 1.706999],accel_mss,speed_ms,0,blend_radius_m)
    |   movel([0.136326, -1.410726, -2.548789, -0.752874, 1.570796, 1.707122],accel_mss,speed_ms,0,blend_radius_m)
    |   movel([0.136292, -1.411324, -2.548340, -0.752724, 1.570796, 1.707088],accel_mss,speed_ms,0,blend_radius_m)
    |   movel([0.136035, -1.412285, -2.547618, -0.752486, 1.570796, 1.706831],accel_mss,speed_ms,0,blend_radius_m)
    |   movel([0.135862, -1.412665, -2.547332, -0.752392, 1.570796, 1.706658],accel_mss,speed_ms,0,blend_radius_m)
    |   movel([0.135410, -1.412972, -2.547101, -0.752316, 1.570796, 1.706207],accel_mss,speed_ms,0,blend_radius_m)
    |   movel([0.132283, -1.413271, -2.546875, -0.752242, 1.570796, 1.703079],accel_mss,speed_ms,0,blend_radius_m)
    |   movel([0.130091, -1.413437, -2.546750, -0.752202, 1.570796, 1.700887],accel_mss,speed_ms,0,blend_radius_m)
    |   movel([0.127857, -1.413746, -2.546518, -0.752126, 1.570796, 1.698653],accel_mss,speed_ms,0,blend_radius_m)
    |   movel([0.122098, -1.414883, -2.545659, -0.751848, 1.570796, 1.692894],accel_mss,speed_ms,0,blend_radius_m)
    |   movel([0.116206, -1.416399, -2.544510, -0.751480, 1.570796, 1.687002],accel_mss,speed_ms,0,blend_radius_m)
    |   movel([0.113761, -1.417160, -2.543933, -0.751296, 1.570796, 1.684557],accel_mss,speed_ms,0,blend_radius_m)
    |   movel([0.106352, -1.419944, -2.541812, -0.750633, 1.570796, 1.677149],accel_mss,speed_ms,0,blend_radius_m)
    |   movel([0.105057, -1.420313, -2.541530, -0.750546, 1.570796, 1.675853],accel_mss,speed_ms,0,blend_radius_m)
    |   movel([0.104722, -1.420296, -2.541543, -0.750550, 1.570796, 1.675519],accel_mss,speed_ms,0,blend_radius_m)
    |   movel([0.104506, -1.420122, -2.541676, -0.750591, 1.570796, 1.675302],accel_mss,speed_ms,0,blend_radius_m)
    |   movel([0.104317, -1.419327, -2.542283, -0.750779, 1.570796, 1.675113],accel_mss,speed_ms,0,blend_radius_m)
    |   movel([0.104380, -1.418600, -2.542837, -0.750952, 1.570796, 1.675176],accel_mss,speed_ms,0,blend_radius_m)
    |   movel([0.104579, -1.418125, -2.543199, -0.751065, 1.570796, 1.675375],accel_mss,speed_ms,0,blend_radius_m)
    |   movel([0.104975, -1.417723, -2.543505, -0.751161, 1.570796, 1.675771],accel_mss,speed_ms,0,blend_radius_m)
    |   movel([0.105717, -1.417253, -2.543862, -0.751274, 1.570796, 1.676514],accel_mss,speed_ms,0,blend_radius_m)
    |   movel([0.108963, -1.415605, -2.545112, -0.751672, 1.570796, 1.679759],accel_mss,speed_ms,0,blend_radius_m)
    |   movel([0.112269, -1.414275, -2.546118, -0.751996, 1.570796, 1.683065],accel_mss,speed_ms,0,blend_radius_m)
    |   movel([0.116520, -1.412896, -2.547158, -0.752335, 1.570796, 1.687316],accel_mss,speed_ms,0,blend_radius_m)
    |   movel([0.120763, -1.411742, -2.548027, -0.752621, 1.570796, 1.691560],accel_mss,speed_ms,0,blend_radius_m)
    |   movel([0.124985, -1.410815, -2.548723, -0.752852, 1.570796, 1.695781],accel_mss,speed_ms,0,blend_radius_m)
    |   movel([0.129158, -1.410124, -2.549240, -0.753024, 1.570796, 1.699955],accel_mss,speed_ms,0,blend_radius_m)
    |   movel([0.132351, -1.409861, -2.549438, -0.753091, 1.570796, 1.703147],accel_mss,speed_ms,0,blend_radius_m)
    |   movel([0.135389, -1.409972, -2.549355, -0.753063, 1.570796, 1.706186],accel_mss,speed_ms,0,blend_radius_m)
    |   movel([0.135900, -1.410093, -2.549263, -0.753032, 1.570796, 1.706696],accel_mss,speed_ms,0,blend_radius_m)
    |   movel([0.136203, -1.410331, -2.549085, -0.752973, 1.570796, 1.706999],accel_mss,speed_ms,0,blend_radius_m)
    |   movel([0.136326, -1.410726, -2.548789, -0.752874, 1.570796, 1.707122],accel_mss,speed_ms,0,blend_radius_m)
    |   movel([0.136292, -1.411324, -2.548340, -0.752724, 1.570796, 1.707088],accel_mss,speed_ms,0,blend_radius_m)
    |   speed_ms = 0.005
    |   movel([0.136292, -1.402874, -2.544470, -0.765045, 1.570796, 1.707088],accel_mss,speed_ms,0,blend_radius_m)
    |   speed_ms = 0.040
    |   movel([0.122958, -1.385670, -2.557008, -0.769711, 1.570796, 1.693754],accel_mss,speed_ms,0,blend_radius_m)
    |   speed_ms = 0.005
    |   movel([0.122958, -1.394244, -2.560951, -0.757194, 1.570796, 1.693754],accel_mss,speed_ms,0,blend_radius_m)
    |   speed_ms = 0.035
    |   movel([0.113172, -1.396655, -2.559197, -0.756537, 1.570796, 1.683968],accel_mss,speed_ms,0,blend_radius_m)
    |   movel([0.109978, -1.397379, -2.558669, -0.756341, 1.570796, 1.680775],accel_mss,speed_ms,0,blend_radius_m)
    |   movel([0.109786, -1.397239, -2.558771, -0.756379, 1.570796, 1.680582],accel_mss,speed_ms,0,blend_radius_m)
    |   movel([0.110029, -1.396984, -2.558957, -0.756448, 1.570796, 1.680825],accel_mss,speed_ms,0,blend_radius_m)
    |   movel([0.117381, -1.394873, -2.560495, -0.757021, 1.570796, 1.688177],accel_mss,speed_ms,0,blend_radius_m)
    |   movel([0.123079, -1.393389, -2.561572, -0.757429, 1.570796, 1.693875],accel_mss,speed_ms,0,blend_radius_m)
    |   movel([0.132890, -1.391039, -2.563270, -0.758080, 1.570796, 1.703686],accel_mss,speed_ms,0,blend_radius_m)
    |   movel([0.136095, -1.390365, -2.563756, -0.758268, 1.570796, 1.706892],accel_mss,speed_ms,0,blend_radius_m)
    |   movel([0.136283, -1.390512, -2.563650, -0.758227, 1.570796, 1.707079],accel_mss,speed_ms,0,blend_radius_m)
    |   movel([0.136033, -1.390766, -2.563467, -0.758156, 1.570796, 1.706829],accel_mss,speed_ms,0,blend_radius_m)
    |   movel([0.128656, -1.392785, -2.562009, -0.757595, 1.570796, 1.699453],accel_mss,speed_ms,0,blend_radius_m)
    |   movel([0.122958, -1.394244, -2.560951, -0.757194, 1.570796, 1.693754],accel_mss,speed_ms,0,blend_radius_m)
    |   movel([0.120510, -1.394841, -2.560518, -0.757030, 1.570796, 1.691306],accel_mss,speed_ms,0,blend_radius_m)
    |   speed_ms = 0.005
    |   movel([0.120510, -1.386271, -2.556577, -0.769541, 1.570796, 1.691306],accel_mss,speed_ms,0,blend_radius_m)
    |   speed_ms = 0.040
    |   movel([0.123568, -1.383020, -2.558901, -0.770467, 1.570796, 1.694365],accel_mss,speed_ms,0,blend_radius_m)
    |   speed_ms = 0.005
    |   movel([0.123568, -1.391613, -2.562856, -0.757920, 1.570796, 1.694365],accel_mss,speed_ms,0,blend_radius_m)
    |   speed_ms = 0.035
    |   movel([0.163298, -1.382075, -2.569677, -0.760637, 1.570796, 1.734095],accel_mss,speed_ms,0,blend_radius_m)
    |   movel([0.171306, -1.339584, -2.598492, -0.774313, 1.570796, 1.742102],accel_mss,speed_ms,0,blend_radius_m)
    |   movel([0.180166, -1.294050, -2.626637, -0.791702, 1.570796, 1.750963],accel_mss,speed_ms,0,blend_radius_m)
    |   movel([0.136190, -1.306028, -2.619498, -0.786863, 1.570796, 1.706987],accel_mss,speed_ms,0,blend_radius_m)
    |   movel([0.092605, -1.319237, -2.611408, -0.781743, 1.570796, 1.663401],accel_mss,speed_ms,0,blend_radius_m)
    |   movel([0.088158, -1.362012, -2.583598, -0.766779, 1.570796, 1.658955],accel_mss,speed_ms,0,blend_radius_m)
    |   movel([0.084125, -1.402203, -2.555128, -0.755058, 1.570796, 1.654922],accel_mss,speed_ms,0,blend_radius_m)
    |   movel([0.123568, -1.391613, -2.562856, -0.757920, 1.570796, 1.694365],accel_mss,speed_ms,0,blend_radius_m)
    |   movel([0.126029, -1.390989, -2.563307, -0.758094, 1.570796, 1.696825],accel_mss,speed_ms,0,blend_radius_m)
    |   speed_ms = 0.005
    |   movel([0.126029, -1.382392, -2.559349, -0.770648, 1.570796, 1.696825],accel_mss,speed_ms,0,blend_radius_m)
    |   speed_ms = 0.040
    |   movel([0.116105, -1.389810, -2.554030, -0.768549, 1.570796, 1.686902],accel_mss,speed_ms,0,blend_radius_m)
    |   speed_ms = 0.005
    |   movel([0.116105, -1.398354, -2.557956, -0.756079, 1.570796, 1.686902],accel_mss,speed_ms,0,blend_radius_m)
    |   speed_ms = 0.035
    |   movel([0.115433, -1.398483, -2.557862, -0.756045, 1.570796, 1.686229],accel_mss,speed_ms,0,blend_radius_m)
    |   movel([0.130214, -1.394704, -2.560618, -0.757068, 1.570796, 1.701011],accel_mss,speed_ms,0,blend_radius_m)
    |   movel([0.126246, -1.395821, -2.559805, -0.756763, 1.570796, 1.697043],accel_mss,speed_ms,0,blend_radius_m)
    |   movel([0.122632, -1.396742, -2.559134, -0.756513, 1.570796, 1.693428],accel_mss,speed_ms,0,blend_radius_m)
    |   movel([0.116105, -1.398354, -2.557956, -0.756079, 1.570796, 1.686902],accel_mss,speed_ms,0,blend_radius_m)
    |   movel([0.115433, -1.398483, -2.557862, -0.756045, 1.570796, 1.686229],accel_mss,speed_ms,0,blend_radius_m)
    |   movel([0.117195, -1.398023, -2.558198, -0.756168, 1.570796, 1.687991],accel_mss,speed_ms,0,blend_radius_m)
    |   speed_ms = 0.005
    |   movel([0.117195, -1.389476, -2.554271, -0.768642, 1.570796, 1.687991],accel_mss,speed_ms,0,blend_radius_m)
    |   speed_ms = 0.040
    |   movel([0.080369, -1.394995, -2.550266, -0.767129, 1.570796, 1.651165],accel_mss,speed_ms,0,blend_radius_m)
    |   speed_ms = 0.005
    |   movel([0.080369, -1.403502, -2.554169, -0.754718, 1.570796, 1.651165],accel_mss,speed_ms,0,blend_radius_m)
    |   speed_ms = 0.035
    |   movel([0.082668, -1.402565, -2.554861, -0.754963, 1.570796, 1.653464],accel_mss,speed_ms,0,blend_radius_m)
    |   movel([0.083132, -1.397781, -2.558375, -0.756233, 1.570796, 1.653929],accel_mss,speed_ms,0,blend_radius_m)
    |   movel([0.083285, -1.395945, -2.559715, -0.756729, 1.570796, 1.654081],accel_mss,speed_ms,0,blend_radius_m)
    |   movel([0.083369, -1.393143, -2.561750, -0.757496, 1.570796, 1.654165],accel_mss,speed_ms,0,blend_radius_m)
    |   movel([0.071293, -1.395474, -2.560058, -0.756858, 1.570796, 1.642090],accel_mss,speed_ms,0,blend_radius_m)
    |   movel([0.066805, -1.396417, -2.559371, -0.756601, 1.570796, 1.637601],accel_mss,speed_ms,0,blend_radius_m)
    |   movel([0.059543, -1.398103, -2.558140, -0.756146, 1.570796, 1.630340],accel_mss,speed_ms,0,blend_radius_m)
    |   movel([0.058947, -1.398356, -2.557954, -0.756078, 1.570796, 1.629743],accel_mss,speed_ms,0,blend_radius_m)
    |   movel([0.058527, -1.398722, -2.557686, -0.755980, 1.570796, 1.629324],accel_mss,speed_ms,0,blend_radius_m)
    |   movel([0.058288, -1.399166, -2.557362, -0.755862, 1.570796, 1.629084],accel_mss,speed_ms,0,blend_radius_m)
    |   movel([0.058040, -1.400671, -2.556256, -0.755462, 1.570796, 1.628837],accel_mss,speed_ms,0,blend_radius_m)
    |   movel([0.058173, -1.402295, -2.555061, -0.755034, 1.570796, 1.628969],accel_mss,speed_ms,0,blend_radius_m)
    |   movel([0.058390, -1.402968, -2.554564, -0.754857, 1.570796, 1.629186],accel_mss,speed_ms,0,blend_radius_m)
    |   movel([0.058721, -1.403569, -2.554119, -0.754700, 1.570796, 1.629517],accel_mss,speed_ms,0,blend_radius_m)
    |   movel([0.059262, -1.404189, -2.553661, -0.754539, 1.570796, 1.630058],accel_mss,speed_ms,0,blend_radius_m)
    |   movel([0.059943, -1.404684, -2.553294, -0.754411, 1.570796, 1.630739],accel_mss,speed_ms,0,blend_radius_m)
    |   movel([0.060908, -1.405173, -2.552932, -0.754285, 1.570796, 1.631705],accel_mss,speed_ms,0,blend_radius_m)
    |   movel([0.061951, -1.405568, -2.552638, -0.754183, 1.570796, 1.632747],accel_mss,speed_ms,0,blend_radius_m)
    |   movel([0.064429, -1.406135, -2.552217, -0.754037, 1.570796, 1.635225],accel_mss,speed_ms,0,blend_radius_m)
    |   movel([0.065734, -1.406268, -2.552118, -0.754003, 1.570796, 1.636530],accel_mss,speed_ms,0,blend_radius_m)
    |   movel([0.068559, -1.406226, -2.552150, -0.754014, 1.570796, 1.639356],accel_mss,speed_ms,0,blend_radius_m)
    |   movel([0.070060, -1.406057, -2.552275, -0.754057, 1.570796, 1.640856],accel_mss,speed_ms,0,blend_radius_m)
    |   movel([0.073745, -1.405404, -2.552760, -0.754225, 1.570796, 1.644541],accel_mss,speed_ms,0,blend_radius_m)
    |   movel([0.077424, -1.404510, -2.553423, -0.754456, 1.570796, 1.648221],accel_mss,speed_ms,0,blend_radius_m)
    |   movel([0.080369, -1.403502, -2.554169, -0.754718, 1.570796, 1.651165],accel_mss,speed_ms,0,blend_radius_m)
    |   movel([0.082668, -1.402565, -2.554861, -0.754963, 1.570796, 1.653464],accel_mss,speed_ms,0,blend_radius_m)
    |   speed_ms = 0.005
    |   movel([0.082679, -1.393931, -2.551041, -0.767417, 1.570796, 1.653475],accel_mss,speed_ms,0,blend_radius_m)
    |   speed_ms = 0.040
    |   movel([0.064626, -1.387514, -2.555685, -0.769190, 1.570796, 1.635422],accel_mss,speed_ms,0,blend_radius_m)
    |   speed_ms = 0.005
    |   movel([0.064626, -1.396075, -2.559620, -0.756694, 1.570796, 1.635422],accel_mss,speed_ms,0,blend_radius_m)
    |   speed_ms = 0.035
    |   movel([0.058998, -1.397165, -2.558825, -0.756399, 1.570796, 1.629795],accel_mss,speed_ms,0,blend_radius_m)
    |   movel([0.059184, -1.396955, -2.558978, -0.756456, 1.570796, 1.629980],accel_mss,speed_ms,0,blend_radius_m)
    |   movel([0.060872, -1.396524, -2.559293, -0.756572, 1.570796, 1.631668],accel_mss,speed_ms,0,blend_radius_m)
    |   movel([0.067359, -1.395085, -2.560340, -0.756963, 1.570796, 1.638155],accel_mss,speed_ms,0,blend_radius_m)
    |   movel([0.069209, -1.394741, -2.560591, -0.757058, 1.570796, 1.640005],accel_mss,speed_ms,0,blend_radius_m)
    |   movel([0.070745, -1.394482, -2.560779, -0.757128, 1.570796, 1.641541],accel_mss,speed_ms,0,blend_radius_m)
    |   movel([0.070556, -1.394692, -2.560626, -0.757071, 1.570796, 1.641353],accel_mss,speed_ms,0,blend_radius_m)
    |   movel([0.068867, -1.395111, -2.560322, -0.756956, 1.570796, 1.639663],accel_mss,speed_ms,0,blend_radius_m)
    |   movel([0.064626, -1.396075, -2.559620, -0.756694, 1.570796, 1.635422],accel_mss,speed_ms,0,blend_radius_m)
    |   movel([0.062208, -1.396540, -2.559281, -0.756568, 1.570796, 1.633005],accel_mss,speed_ms,0,blend_radius_m)
    |   speed_ms = 0.005
    |   movel([0.062208, -1.387983, -2.555347, -0.769059, 1.570796, 1.633005],accel_mss,speed_ms,0,blend_radius_m)
    |   speed_ms = 0.040
    |   movel([0.077329, -1.384953, -2.557521, -0.769914, 1.570796, 1.648125],accel_mss,speed_ms,0,blend_radius_m)
    |   speed_ms = 0.005
    |   movel([0.077329, -1.393532, -2.561468, -0.757389, 1.570796, 1.648125],accel_mss,speed_ms,0,blend_radius_m)
    |   speed_ms = 0.035
    |   movel([0.071698, -1.394568, -2.560716, -0.757105, 1.570796, 1.642495],accel_mss,speed_ms,0,blend_radius_m)
    |   movel([0.071887, -1.394358, -2.560869, -0.757162, 1.570796, 1.642683],accel_mss,speed_ms,0,blend_radius_m)
    |   movel([0.073577, -1.393942, -2.561170, -0.757276, 1.570796, 1.644374],accel_mss,speed_ms,0,blend_radius_m)
    |   movel([0.080071, -1.392565, -2.562168, -0.757656, 1.570796, 1.650867],accel_mss,speed_ms,0,blend_radius_m)
    |   movel([0.081921, -1.392238, -2.562404, -0.757746, 1.570796, 1.652718],accel_mss,speed_ms,0,blend_radius_m)
    |   movel([0.083457, -1.391995, -2.562580, -0.757814, 1.570796, 1.654253],accel_mss,speed_ms,0,blend_radius_m)
    |   movel([0.083266, -1.392204, -2.562429, -0.757756, 1.570796, 1.654062],accel_mss,speed_ms,0,blend_radius_m)
    |   movel([0.081574, -1.392608, -2.562137, -0.757644, 1.570796, 1.652370],accel_mss,speed_ms,0,blend_radius_m)
    |   movel([0.077329, -1.393532, -2.561468, -0.757389, 1.570796, 1.648125],accel_mss,speed_ms,0,blend_radius_m)
    |   movel([0.074910, -1.393974, -2.561147, -0.757268, 1.570796, 1.645706],accel_mss,speed_ms,0,blend_radius_m)
    |   speed_ms = 0.005
    |   movel([0.074910, -1.385398, -2.557203, -0.769788, 1.570796, 1.645706],accel_mss,speed_ms,0,blend_radius_m)
    |   speed_ms = 0.040
    |   movel([0.082596, -1.382598, -2.559202, -0.770589, 1.570796, 1.653392],accel_mss,speed_ms,0,blend_radius_m)
    |   speed_ms = 0.005
    |   movel([0.082596, -1.391193, -2.563159, -0.758037, 1.570796, 1.653392],accel_mss,speed_ms,0,blend_radius_m)
    |   speed_ms = 0.035
    |   movel([0.080067, -1.391807, -2.562716, -0.757866, 1.570796, 1.650864],accel_mss,speed_ms,0,blend_radius_m)
    |   movel([0.070347, -1.393735, -2.561320, -0.757333, 1.570796, 1.641143],accel_mss,speed_ms,0,blend_radius_m)
    |   movel([0.059849, -1.395878, -2.559764, -0.756748, 1.570796, 1.630646],accel_mss,speed_ms,0,blend_radius_m)
    |   movel([0.059405, -1.395830, -2.559798, -0.756761, 1.570796, 1.630201],accel_mss,speed_ms,0,blend_radius_m)
    |   movel([0.059560, -1.395474, -2.560058, -0.756857, 1.570796, 1.630356],accel_mss,speed_ms,0,blend_radius_m)
    |   movel([0.061171, -1.394941, -2.560445, -0.757003, 1.570796, 1.631968],accel_mss,speed_ms,0,blend_radius_m)
    |   movel([0.064490, -1.394119, -2.561042, -0.757228, 1.570796, 1.635287],accel_mss,speed_ms,0,blend_radius_m)
    |   movel([0.083770, -1.390021, -2.564003, -0.758364, 1.570796, 1.654566],accel_mss,speed_ms,0,blend_radius_m)
    |   movel([0.083851, -1.390419, -2.563717, -0.758253, 1.570796, 1.654647],accel_mss,speed_ms,0,blend_radius_m)
    |   movel([0.083064, -1.391027, -2.563279, -0.758083, 1.570796, 1.653860],accel_mss,speed_ms,0,blend_radius_m)
    |   movel([0.082596, -1.391193, -2.563159, -0.758037, 1.570796, 1.653392],accel_mss,speed_ms,0,blend_radius_m)
    |   movel([0.080141, -1.391789, -2.562729, -0.757871, 1.570796, 1.650937],accel_mss,speed_ms,0,blend_radius_m)
    |   speed_ms = 0.005
    |   movel([0.080141, -1.383198, -2.558775, -0.770416, 1.570796, 1.650937],accel_mss,speed_ms,0,blend_radius_m)
    |   speed_ms = 0.040
    |   movel([0.080979, -1.380162, -2.560933, -0.771295, 1.570796, 1.651775],accel_mss,speed_ms,0,blend_radius_m)
    |   speed_ms = 0.005
    |   movel([0.080979, -1.388774, -2.564900, -0.758715, 1.570796, 1.651775],accel_mss,speed_ms,0,blend_radius_m)
    |   speed_ms = 0.035
    |   movel([0.077024, -1.389691, -2.564241, -0.758457, 1.570796, 1.647820],accel_mss,speed_ms,0,blend_radius_m)
    |   movel([0.073579, -1.390441, -2.563701, -0.758247, 1.570796, 1.644375],accel_mss,speed_ms,0,blend_radius_m)
    |   movel([0.059877, -1.393440, -2.561534, -0.757414, 1.570796, 1.630673],accel_mss,speed_ms,0,blend_radius_m)
    |   movel([0.060254, -1.384100, -2.568239, -0.760049, 1.570796, 1.631050],accel_mss,speed_ms,0,blend_radius_m)
    |   movel([0.060698, -1.378163, -2.572436, -0.761790, 1.570796, 1.631494],accel_mss,speed_ms,0,blend_radius_m)
    |   movel([0.061960, -1.362407, -2.583329, -0.766652, 1.570796, 1.632757],accel_mss,speed_ms,0,blend_radius_m)
    |   movel([0.073910, -1.358507, -2.585972, -0.767910, 1.570796, 1.644706],accel_mss,speed_ms,0,blend_radius_m)
    |   movel([0.085905, -1.354690, -2.588537, -0.769162, 1.570796, 1.656701],accel_mss,speed_ms,0,blend_radius_m)
    |   movel([0.084226, -1.371704, -2.576944, -0.763740, 1.570796, 1.655023],accel_mss,speed_ms,0,blend_radius_m)
    |   movel([0.082613, -1.388299, -2.565241, -0.758849, 1.570796, 1.653409],accel_mss,speed_ms,0,blend_radius_m)
    |   movel([0.080979, -1.388774, -2.564900, -0.758715, 1.570796, 1.651775],accel_mss,speed_ms,0,blend_radius_m)
    |   movel([0.078522, -1.389342, -2.564492, -0.758555, 1.570796, 1.649318],accel_mss,speed_ms,0,blend_radius_m)
    |   speed_ms = 0.005
    |   movel([0.078522, -1.380733, -2.560527, -0.771128, 1.570796, 1.649318],accel_mss,speed_ms,0,blend_radius_m)
    |   speed_ms = 0.040
    |   movel([0.104255, -1.353104, -2.579589, -0.779697, 1.570796, 1.675051],accel_mss,speed_ms,0,blend_radius_m)
    |   speed_ms = 0.005
    |   movel([0.104255, -1.361901, -2.583674, -0.766814, 1.570796, 1.675051],accel_mss,speed_ms,0,blend_radius_m)
    |   speed_ms = 0.035
    |   movel([0.103098, -1.361251, -2.584115, -0.767023, 1.570796, 1.673894],accel_mss,speed_ms,0,blend_radius_m)
    |   movel([0.102445, -1.361066, -2.584241, -0.767082, 1.570796, 1.673242],accel_mss,speed_ms,0,blend_radius_m)
    |   movel([0.101234, -1.361003, -2.584283, -0.767103, 1.570796, 1.672030],accel_mss,speed_ms,0,blend_radius_m)
    |   movel([0.100898, -1.360790, -2.584428, -0.767171, 1.570796, 1.671694],accel_mss,speed_ms,0,blend_radius_m)
    |   movel([0.100780, -1.360314, -2.584750, -0.767325, 1.570796, 1.671576],accel_mss,speed_ms,0,blend_radius_m)
    |   movel([0.100845, -1.359346, -2.585405, -0.767638, 1.570796, 1.671642],accel_mss,speed_ms,0,blend_radius_m)
    |   movel([0.100904, -1.358519, -2.585964, -0.767906, 1.570796, 1.671701],accel_mss,speed_ms,0,blend_radius_m)
    |   movel([0.100827, -1.358027, -2.586296, -0.768066, 1.570796, 1.671624],accel_mss,speed_ms,0,blend_radius_m)
    |   movel([0.100621, -1.357799, -2.586449, -0.768141, 1.570796, 1.671417],accel_mss,speed_ms,0,blend_radius_m)
    |   movel([0.100282, -1.357790, -2.586455, -0.768144, 1.570796, 1.671078],accel_mss,speed_ms,0,blend_radius_m)
    |   movel([0.099917, -1.358002, -2.586313, -0.768075, 1.570796, 1.670713],accel_mss,speed_ms,0,blend_radius_m)
    |   movel([0.099642, -1.358367, -2.586066, -0.767956, 1.570796, 1.670438],accel_mss,speed_ms,0,blend_radius_m)
    |   movel([0.099443, -1.358935, -2.585683, -0.767771, 1.570796, 1.670239],accel_mss,speed_ms,0,blend_radius_m)
    |   movel([0.099310, -1.359772, -2.585117, -0.767500, 1.570796, 1.670106],accel_mss,speed_ms,0,blend_radius_m)
    |   movel([0.099160, -1.360667, -2.584511, -0.767211, 1.570796, 1.669956],accel_mss,speed_ms,0,blend_radius_m)
    |   movel([0.098932, -1.361273, -2.584100, -0.767016, 1.570796, 1.669729],accel_mss,speed_ms,0,blend_radius_m)
    |   movel([0.098585, -1.361720, -2.583796, -0.766872, 1.570796, 1.669381],accel_mss,speed_ms,0,blend_radius_m)
    |   movel([0.098078, -1.362089, -2.583546, -0.766754, 1.570796, 1.668874],accel_mss,speed_ms,0,blend_radius_m)
    |   movel([0.096923, -1.362996, -2.582929, -0.766464, 1.570796, 1.667719],accel_mss,speed_ms,0,blend_radius_m)
    |   movel([0.096227, -1.363675, -2.582466, -0.766248, 1.570796, 1.667024],accel_mss,speed_ms,0,blend_radius_m)
    |   movel([0.095599, -1.364374, -2.581989, -0.766026, 1.570796, 1.666396],accel_mss,speed_ms,0,blend_radius_m)
    |   movel([0.094796, -1.365509, -2.581213, -0.765667, 1.570796, 1.665593],accel_mss,speed_ms,0,blend_radius_m)
    |   movel([0.094259, -1.366681, -2.580410, -0.765299, 1.570796, 1.665056],accel_mss,speed_ms,0,blend_radius_m)
    |   movel([0.094002, -1.367845, -2.579610, -0.764934, 1.570796, 1.664798],accel_mss,speed_ms,0,blend_radius_m)
    |   movel([0.094042, -1.368919, -2.578870, -0.764600, 1.570796, 1.664839],accel_mss,speed_ms,0,blend_radius_m)
    |   movel([0.094371, -1.369840, -2.578234, -0.764314, 1.570796, 1.665168],accel_mss,speed_ms,0,blend_radius_m)
    |   movel([0.094976, -1.370568, -2.577731, -0.764090, 1.570796, 1.665772],accel_mss,speed_ms,0,blend_radius_m)
    |   movel([0.095809, -1.371034, -2.577408, -0.763946, 1.570796, 1.666605],accel_mss,speed_ms,0,blend_radius_m)
    |   movel([0.097424, -1.371338, -2.577198, -0.763853, 1.570796, 1.668221],accel_mss,speed_ms,0,blend_radius_m)
    |   movel([0.097739, -1.371607, -2.577012, -0.763770, 1.570796, 1.668535],accel_mss,speed_ms,0,blend_radius_m)
    |   movel([0.097855, -1.372114, -2.576660, -0.763615, 1.570796, 1.668651],accel_mss,speed_ms,0,blend_radius_m)
    |   movel([0.097799, -1.373040, -2.576016, -0.763332, 1.570796, 1.668595],accel_mss,speed_ms,0,blend_radius_m)
    |   movel([0.097730, -1.373976, -2.575366, -0.763048, 1.570796, 1.668526],accel_mss,speed_ms,0,blend_radius_m)
    |   movel([0.097826, -1.374415, -2.575059, -0.762914, 1.570796, 1.668623],accel_mss,speed_ms,0,blend_radius_m)
    |   movel([0.098103, -1.374573, -2.574949, -0.762867, 1.570796, 1.668900],accel_mss,speed_ms,0,blend_radius_m)
    |   movel([0.098607, -1.374512, -2.574992, -0.762885, 1.570796, 1.669404],accel_mss,speed_ms,0,blend_radius_m)
    |   movel([0.099131, -1.374281, -2.575153, -0.762955, 1.570796, 1.669927],accel_mss,speed_ms,0,blend_radius_m)
    |   movel([0.099463, -1.373955, -2.575380, -0.763054, 1.570796, 1.670260],accel_mss,speed_ms,0,blend_radius_m)
    |   movel([0.099670, -1.373433, -2.575743, -0.763212, 1.570796, 1.670466],accel_mss,speed_ms,0,blend_radius_m)
    |   movel([0.099815, -1.372488, -2.576400, -0.763501, 1.570796, 1.670612],accel_mss,speed_ms,0,blend_radius_m)
    |   movel([0.099987, -1.371509, -2.577080, -0.763800, 1.570796, 1.670783],accel_mss,speed_ms,0,blend_radius_m)
    |   movel([0.100262, -1.370864, -2.577526, -0.763999, 1.570796, 1.671058],accel_mss,speed_ms,0,blend_radius_m)
    |   movel([0.100743, -1.370307, -2.577912, -0.764170, 1.570796, 1.671539],accel_mss,speed_ms,0,blend_radius_m)
    |   movel([0.101583, -1.369654, -2.578363, -0.764372, 1.570796, 1.672379],accel_mss,speed_ms,0,blend_radius_m)
    |   movel([0.102710, -1.368753, -2.578984, -0.764651, 1.570796, 1.673506],accel_mss,speed_ms,0,blend_radius_m)
    |   movel([0.103698, -1.367721, -2.579695, -0.764973, 1.570796, 1.674494],accel_mss,speed_ms,0,blend_radius_m)
    |   movel([0.104455, -1.366649, -2.580432, -0.765309, 1.570796, 1.675251],accel_mss,speed_ms,0,blend_radius_m)
    |   movel([0.104969, -1.365539, -2.581192, -0.765658, 1.570796, 1.675765],accel_mss,speed_ms,0,blend_radius_m)
    |   movel([0.105210, -1.364466, -2.581926, -0.765997, 1.570796, 1.676006],accel_mss,speed_ms,0,blend_radius_m)
    |   movel([0.105164, -1.363480, -2.582599, -0.766310, 1.570796, 1.675960],accel_mss,speed_ms,0,blend_radius_m)
    |   movel([0.104837, -1.362602, -2.583197, -0.766590, 1.570796, 1.675633],accel_mss,speed_ms,0,blend_radius_m)
    |   movel([0.104255, -1.361901, -2.583674, -0.766814, 1.570796, 1.675051],accel_mss,speed_ms,0,blend_radius_m)
    |   movel([0.103098, -1.361251, -2.584115, -0.767023, 1.570796, 1.673894],accel_mss,speed_ms,0,blend_radius_m)
    |   movel([0.102445, -1.361066, -2.584241, -0.767082, 1.570796, 1.673242],accel_mss,speed_ms,0,blend_radius_m)
    |   speed_ms = 0.005
    |   movel([0.102445, -1.352263, -2.580152, -0.779974, 1.570796, 1.673242],accel_mss,speed_ms,0,blend_radius_m)
    |   speed_ms = 0.040
    |   movel([0.122669, -1.347908, -2.583054, -0.781427, 1.570796, 1.693465],accel_mss,speed_ms,0,blend_radius_m)
    |   speed_ms = 0.005
    |   movel([0.122669, -1.356740, -2.587162, -0.768487, 1.570796, 1.693465],accel_mss,speed_ms,0,blend_radius_m)
    |   speed_ms = 0.035
    |   movel([0.123241, -1.357498, -2.586652, -0.768239, 1.570796, 1.694037],accel_mss,speed_ms,0,blend_radius_m)
    |   movel([0.123515, -1.358453, -2.586008, -0.767928, 1.570796, 1.694312],accel_mss,speed_ms,0,blend_radius_m)
    |   movel([0.123489, -1.359567, -2.585256, -0.767566, 1.570796, 1.694285],accel_mss,speed_ms,0,blend_radius_m)
    |   movel([0.123164, -1.360757, -2.584450, -0.767182, 1.570796, 1.693960],accel_mss,speed_ms,0,blend_radius_m)
    |   movel([0.122566, -1.361949, -2.583641, -0.766799, 1.570796, 1.693363],accel_mss,speed_ms,0,blend_radius_m)
    |   movel([0.121723, -1.363092, -2.582863, -0.766434, 1.570796, 1.692519],accel_mss,speed_ms,0,blend_radius_m)
    |   movel([0.120700, -1.364084, -2.582187, -0.766118, 1.570796, 1.691497],accel_mss,speed_ms,0,blend_radius_m)
    |   movel([0.119531, -1.364897, -2.581632, -0.765861, 1.570796, 1.690327],accel_mss,speed_ms,0,blend_radius_m)
    |   movel([0.118876, -1.365355, -2.581318, -0.765716, 1.570796, 1.689673],accel_mss,speed_ms,0,blend_radius_m)
    |   movel([0.118467, -1.365829, -2.580994, -0.765566, 1.570796, 1.689263],accel_mss,speed_ms,0,blend_radius_m)
    |   movel([0.118210, -1.366445, -2.580572, -0.765373, 1.570796, 1.689006],accel_mss,speed_ms,0,blend_radius_m)
    |   movel([0.118030, -1.367413, -2.579907, -0.765069, 1.570796, 1.688826],accel_mss,speed_ms,0,blend_radius_m)
    |   movel([0.117877, -1.368268, -2.579318, -0.764802, 1.570796, 1.688674],accel_mss,speed_ms,0,blend_radius_m)
    |   movel([0.117669, -1.368837, -2.578927, -0.764625, 1.570796, 1.688465],accel_mss,speed_ms,0,blend_radius_m)
    |   movel([0.117391, -1.369198, -2.578678, -0.764513, 1.570796, 1.688187],accel_mss,speed_ms,0,blend_radius_m)
    |   movel([0.117030, -1.369402, -2.578537, -0.764450, 1.570796, 1.687826],accel_mss,speed_ms,0,blend_radius_m)
    |   movel([0.116700, -1.369389, -2.578546, -0.764454, 1.570796, 1.687496],accel_mss,speed_ms,0,blend_radius_m)
    |   movel([0.116500, -1.369169, -2.578698, -0.764522, 1.570796, 1.687297],accel_mss,speed_ms,0,blend_radius_m)
    |   movel([0.116432, -1.368699, -2.579022, -0.764668, 1.570796, 1.687228],accel_mss,speed_ms,0,blend_radius_m)
    |   movel([0.116497, -1.367919, -2.579559, -0.764911, 1.570796, 1.687293],accel_mss,speed_ms,0,blend_radius_m)
    |   movel([0.116560, -1.366975, -2.580208, -0.765206, 1.570796, 1.687356],accel_mss,speed_ms,0,blend_radius_m)
    |   movel([0.116405, -1.366469, -2.580555, -0.765365, 1.570796, 1.687201],accel_mss,speed_ms,0,blend_radius_m)
    |   movel([0.115974, -1.366176, -2.580756, -0.765457, 1.570796, 1.686771],accel_mss,speed_ms,0,blend_radius_m)
    |   movel([0.114418, -1.365819, -2.581001, -0.765570, 1.570796, 1.685215],accel_mss,speed_ms,0,blend_radius_m)
    |   movel([0.113847, -1.365565, -2.581175, -0.765650, 1.570796, 1.684643],accel_mss,speed_ms,0,blend_radius_m)
    |   movel([0.112969, -1.364774, -2.581716, -0.765899, 1.570796, 1.683766],accel_mss,speed_ms,0,blend_radius_m)
    |   movel([0.112679, -1.364249, -2.582074, -0.766066, 1.570796, 1.683475],accel_mss,speed_ms,0,blend_radius_m)
    |   movel([0.112427, -1.363007, -2.582921, -0.766461, 1.570796, 1.683223],accel_mss,speed_ms,0,blend_radius_m)
    |   movel([0.112469, -1.362316, -2.583392, -0.766682, 1.570796, 1.683266],accel_mss,speed_ms,0,blend_radius_m)
    |   movel([0.112890, -1.360876, -2.584369, -0.767143, 1.570796, 1.683686],accel_mss,speed_ms,0,blend_radius_m)
    |   movel([0.113263, -1.360144, -2.584865, -0.767379, 1.570796, 1.684059],accel_mss,speed_ms,0,blend_radius_m)
    |   movel([0.114280, -1.358759, -2.585802, -0.767828, 1.570796, 1.685076],accel_mss,speed_ms,0,blend_radius_m)
    |   movel([0.114910, -1.358133, -2.586224, -0.768032, 1.570796, 1.685707],accel_mss,speed_ms,0,blend_radius_m)
    |   movel([0.116347, -1.357082, -2.586932, -0.768375, 1.570796, 1.687143],accel_mss,speed_ms,0,blend_radius_m)
    |   movel([0.116965, -1.356634, -2.587233, -0.768522, 1.570796, 1.687762],accel_mss,speed_ms,0,blend_radius_m)
    |   movel([0.117363, -1.356155, -2.587555, -0.768679, 1.570796, 1.688160],accel_mss,speed_ms,0,blend_radius_m)
    |   movel([0.117619, -1.355526, -2.587977, -0.768886, 1.570796, 1.688415],accel_mss,speed_ms,0,blend_radius_m)
    |   movel([0.117799, -1.354556, -2.588627, -0.769206, 1.570796, 1.688595],accel_mss,speed_ms,0,blend_radius_m)
    |   movel([0.117970, -1.353565, -2.589290, -0.769534, 1.570796, 1.688766],accel_mss,speed_ms,0,blend_radius_m)
    |   movel([0.118192, -1.353021, -2.589653, -0.769715, 1.570796, 1.688988],accel_mss,speed_ms,0,blend_radius_m)
    |   movel([0.118538, -1.352680, -2.589880, -0.769829, 1.570796, 1.689334],accel_mss,speed_ms,0,blend_radius_m)
    |   movel([0.119076, -1.352445, -2.590036, -0.769907, 1.570796, 1.689873],accel_mss,speed_ms,0,blend_radius_m)
    |   movel([0.119591, -1.352388, -2.590075, -0.769926, 1.570796, 1.690387],accel_mss,speed_ms,0,blend_radius_m)
    |   movel([0.119869, -1.352549, -2.589968, -0.769873, 1.570796, 1.690665],accel_mss,speed_ms,0,blend_radius_m)
    |   movel([0.119956, -1.352998, -2.589668, -0.769723, 1.570796, 1.690753],accel_mss,speed_ms,0,blend_radius_m)
    |   movel([0.119864, -1.353944, -2.589036, -0.769409, 1.570796, 1.690660],accel_mss,speed_ms,0,blend_radius_m)
    |   movel([0.119791, -1.354825, -2.588447, -0.769117, 1.570796, 1.690587],accel_mss,speed_ms,0,blend_radius_m)
    |   movel([0.119877, -1.355347, -2.588097, -0.768945, 1.570796, 1.690674],accel_mss,speed_ms,0,blend_radius_m)
    |   movel([0.120136, -1.355626, -2.587910, -0.768853, 1.570796, 1.690932],accel_mss,speed_ms,0,blend_radius_m)
    |   movel([0.121035, -1.355796, -2.587796, -0.768797, 1.570796, 1.691831],accel_mss,speed_ms,0,blend_radius_m)
    |   movel([0.121598, -1.356026, -2.587641, -0.768721, 1.570796, 1.692395],accel_mss,speed_ms,0,blend_radius_m)
    |   movel([0.122669, -1.356740, -2.587162, -0.768487, 1.570796, 1.693465],accel_mss,speed_ms,0,blend_radius_m)
    |   movel([0.123241, -1.357498, -2.586652, -0.768239, 1.570796, 1.694037],accel_mss,speed_ms,0,blend_radius_m)
    |   movel([0.123512, -1.358441, -2.586016, -0.767932, 1.570796, 1.694308],accel_mss,speed_ms,0,blend_radius_m)
    |   speed_ms = 0.005
    |   movel([0.123512, -1.349620, -2.581916, -0.780852, 1.570796, 1.694308],accel_mss,speed_ms,0,blend_radius_m)
    |   speed_ms = 0.040
    |   movel([0.153851, -1.353048, -2.579626, -0.779715, 1.570796, 1.724647],accel_mss,speed_ms,0,blend_radius_m)
    |   speed_ms = 0.005
    |   movel([0.153851, -1.361846, -2.583711, -0.766832, 1.570796, 1.724647],accel_mss,speed_ms,0,blend_radius_m)
    |   speed_ms = 0.035
    |   movel([0.154055, -1.361944, -2.583645, -0.766801, 1.570796, 1.724851],accel_mss,speed_ms,0,blend_radius_m)
    |   movel([0.154117, -1.362158, -2.583499, -0.766732, 1.570796, 1.724914],accel_mss,speed_ms,0,blend_radius_m)
    |   movel([0.153921, -1.364175, -2.582125, -0.766089, 1.570796, 1.724717],accel_mss,speed_ms,0,blend_radius_m)
    |   movel([0.152612, -1.372455, -2.576424, -0.763511, 1.570796, 1.723408],accel_mss,speed_ms,0,blend_radius_m)
    |   movel([0.150820, -1.382832, -2.569140, -0.760417, 1.570796, 1.721617],accel_mss,speed_ms,0,blend_radius_m)
    |   movel([0.149665, -1.383335, -2.568783, -0.760271, 1.570796, 1.720461],accel_mss,speed_ms,0,blend_radius_m)
    |   movel([0.148775, -1.383636, -2.568569, -0.760184, 1.570796, 1.719571],accel_mss,speed_ms,0,blend_radius_m)
    |   movel([0.122595, -1.390113, -2.563938, -0.758339, 1.570796, 1.693391],accel_mss,speed_ms,0,blend_radius_m)
    |   movel([0.096796, -1.396842, -2.559061, -0.756486, 1.570796, 1.667592],accel_mss,speed_ms,0,blend_radius_m)
    |   movel([0.097952, -1.386630, -2.566436, -0.759323, 1.570796, 1.668749],accel_mss,speed_ms,0,blend_radius_m)
    |   movel([0.099137, -1.376260, -2.573770, -0.762358, 1.570796, 1.669934],accel_mss,speed_ms,0,blend_radius_m)
    |   movel([0.145446, -1.363804, -2.582378, -0.766207, 1.570796, 1.716242],accel_mss,speed_ms,0,blend_radius_m)
    |   movel([0.153343, -1.361886, -2.583684, -0.766819, 1.570796, 1.724139],accel_mss,speed_ms,0,blend_radius_m)
    |   movel([0.153851, -1.361846, -2.583711, -0.766832, 1.570796, 1.724647],accel_mss,speed_ms,0,blend_radius_m)
    |   movel([0.154055, -1.361944, -2.583645, -0.766801, 1.570796, 1.724851],accel_mss,speed_ms,0,blend_radius_m)
    |   movel([0.154117, -1.362158, -2.583499, -0.766732, 1.570796, 1.724914],accel_mss,speed_ms,0,blend_radius_m)
    |   movel([0.153951, -1.363865, -2.582336, -0.766188, 1.570796, 1.724747],accel_mss,speed_ms,0,blend_radius_m)
    |   speed_ms = 0.005
    |   movel([0.153951, -1.355081, -2.578260, -0.779048, 1.570796, 1.724747],accel_mss,speed_ms,0,blend_radius_m)
    |   speed_ms = 0.040
    |   movel([0.189787, -1.362419, -2.573282, -0.776689, 1.570796, 1.760584],accel_mss,speed_ms,0,blend_radius_m)
    |   speed_ms = 0.005
    |   movel([0.189787, -1.371154, -2.577326, -0.763910, 1.570796, 1.760584],accel_mss,speed_ms,0,blend_radius_m)
    |   speed_ms = 0.035
    |   movel([0.190802, -1.369968, -2.578146, -0.764275, 1.570796, 1.761598],accel_mss,speed_ms,0,blend_radius_m)
    |   movel([0.191525, -1.368921, -2.578869, -0.764599, 1.570796, 1.762322],accel_mss,speed_ms,0,blend_radius_m)
    |   movel([0.192069, -1.367827, -2.579622, -0.764940, 1.570796, 1.762865],accel_mss,speed_ms,0,blend_radius_m)
    |   movel([0.192539, -1.366501, -2.580533, -0.765355, 1.570796, 1.763335],accel_mss,speed_ms,0,blend_radius_m)
    |   movel([0.192725, -1.365663, -2.581108, -0.765619, 1.570796, 1.763521],accel_mss,speed_ms,0,blend_radius_m)
    |   movel([0.192760, -1.364863, -2.581654, -0.765871, 1.570796, 1.763557],accel_mss,speed_ms,0,blend_radius_m)
    |   movel([0.192564, -1.364494, -2.581907, -0.765988, 1.570796, 1.763360],accel_mss,speed_ms,0,blend_radius_m)
    |   movel([0.192094, -1.364404, -2.581969, -0.766017, 1.570796, 1.762890],accel_mss,speed_ms,0,blend_radius_m)
    |   movel([0.190038, -1.364853, -2.581662, -0.765874, 1.570796, 1.760834],accel_mss,speed_ms,0,blend_radius_m)
    |   movel([0.178831, -1.368331, -2.579275, -0.764783, 1.570796, 1.749628],accel_mss,speed_ms,0,blend_radius_m)
    |   movel([0.166819, -1.372170, -2.576621, -0.763598, 1.570796, 1.737615],accel_mss,speed_ms,0,blend_radius_m)
    |   movel([0.165845, -1.376607, -2.573528, -0.762254, 1.570796, 1.736641],accel_mss,speed_ms,0,blend_radius_m)
    |   movel([0.165504, -1.378321, -2.572325, -0.761743, 1.570796, 1.736300],accel_mss,speed_ms,0,blend_radius_m)
    |   movel([0.165157, -1.381024, -2.570420, -0.760945, 1.570796, 1.735953],accel_mss,speed_ms,0,blend_radius_m)
    |   movel([0.165274, -1.381323, -2.570209, -0.760857, 1.570796, 1.736070],accel_mss,speed_ms,0,blend_radius_m)
    |   movel([0.165728, -1.381529, -2.570063, -0.760797, 1.570796, 1.736525],accel_mss,speed_ms,0,blend_radius_m)
    |   movel([0.166306, -1.381544, -2.570053, -0.760793, 1.570796, 1.737103],accel_mss,speed_ms,0,blend_radius_m)
    |   movel([0.169378, -1.381033, -2.570414, -0.760942, 1.570796, 1.740174],accel_mss,speed_ms,0,blend_radius_m)
    |   movel([0.172884, -1.380232, -2.570980, -0.761178, 1.570796, 1.743681],accel_mss,speed_ms,0,blend_radius_m)
    |   movel([0.176221, -1.379217, -2.571695, -0.761477, 1.570796, 1.747017],accel_mss,speed_ms,0,blend_radius_m)
    |   movel([0.178197, -1.378476, -2.572216, -0.761697, 1.570796, 1.748994],accel_mss,speed_ms,0,blend_radius_m)
    |   movel([0.180168, -1.377623, -2.572815, -0.761951, 1.570796, 1.750964],accel_mss,speed_ms,0,blend_radius_m)
    |   movel([0.182082, -1.376676, -2.573480, -0.762234, 1.570796, 1.752878],accel_mss,speed_ms,0,blend_radius_m)
    |   movel([0.183972, -1.375617, -2.574220, -0.762552, 1.570796, 1.754769],accel_mss,speed_ms,0,blend_radius_m)
    |   movel([0.185660, -1.374555, -2.574962, -0.762872, 1.570796, 1.756456],accel_mss,speed_ms,0,blend_radius_m)
    |   movel([0.187300, -1.373394, -2.575771, -0.763224, 1.570796, 1.758096],accel_mss,speed_ms,0,blend_radius_m)
    |   movel([0.188599, -1.372327, -2.576512, -0.763550, 1.570796, 1.759395],accel_mss,speed_ms,0,blend_radius_m)
    |   movel([0.189787, -1.371154, -2.577326, -0.763910, 1.570796, 1.760584],accel_mss,speed_ms,0,blend_radius_m)
    |   movel([0.190802, -1.369968, -2.578146, -0.764275, 1.570796, 1.761598],accel_mss,speed_ms,0,blend_radius_m)
    |   movel([0.191494, -1.368966, -2.578838, -0.764585, 1.570796, 1.762290],accel_mss,speed_ms,0,blend_radius_m)
    |   speed_ms = 0.005
    |   movel([0.191494, -1.360216, -2.574784, -0.777389, 1.570796, 1.762290],accel_mss,speed_ms,0,blend_radius_m)
    |   speed_ms = 0.040
    |   movel([0.192479, -1.354542, -2.578623, -0.779224, 1.570796, 1.763275],accel_mss,speed_ms,0,blend_radius_m)
    |   speed_ms = 0.005
    |   movel([0.192479, -1.363330, -2.582701, -0.766358, 1.570796, 1.763275],accel_mss,speed_ms,0,blend_radius_m)
    |   speed_ms = 0.035
    |   movel([0.172891, -1.369439, -2.578512, -0.764439, 1.570796, 1.743688],accel_mss,speed_ms,0,blend_radius_m)
    |   movel([0.168962, -1.370537, -2.577753, -0.764099, 1.570796, 1.739758],accel_mss,speed_ms,0,blend_radius_m)
    |   movel([0.167006, -1.370884, -2.577512, -0.763992, 1.570796, 1.737802],accel_mss,speed_ms,0,blend_radius_m)
    |   movel([0.166803, -1.370755, -2.577602, -0.764032, 1.570796, 1.737599],accel_mss,speed_ms,0,blend_radius_m)
    |   movel([0.166931, -1.370466, -2.577802, -0.764121, 1.570796, 1.737728],accel_mss,speed_ms,0,blend_radius_m)
    |   movel([0.167353, -1.370216, -2.577975, -0.764198, 1.570796, 1.738149],accel_mss,speed_ms,0,blend_radius_m)
    |   movel([0.190050, -1.363047, -2.582894, -0.766448, 1.570796, 1.760846],accel_mss,speed_ms,0,blend_radius_m)
    |   movel([0.192176, -1.362501, -2.583266, -0.766622, 1.570796, 1.762972],accel_mss,speed_ms,0,blend_radius_m)
    |   movel([0.192671, -1.362514, -2.583257, -0.766618, 1.570796, 1.763467],accel_mss,speed_ms,0,blend_radius_m)
    |   movel([0.192945, -1.362770, -2.583082, -0.766536, 1.570796, 1.763742],accel_mss,speed_ms,0,blend_radius_m)
    |   movel([0.192847, -1.363094, -2.582862, -0.766433, 1.570796, 1.763643],accel_mss,speed_ms,0,blend_radius_m)
    |   movel([0.192479, -1.363330, -2.582701, -0.766358, 1.570796, 1.763275],accel_mss,speed_ms,0,blend_radius_m)
    |   movel([0.189922, -1.364113, -2.582167, -0.766109, 1.570796, 1.760718],accel_mss,speed_ms,0,blend_radius_m)
    |   speed_ms = 0.005
    |   movel([0.189922, -1.355331, -2.578092, -0.778967, 1.570796, 1.760718],accel_mss,speed_ms,0,blend_radius_m)
    |   speed_ms = 0.040
    |   movel([0.190579, -1.353295, -2.579461, -0.779634, 1.570796, 1.761375],accel_mss,speed_ms,0,blend_radius_m)
    |   speed_ms = 0.005
    |   movel([0.190579, -1.362091, -2.583545, -0.766753, 1.570796, 1.761375],accel_mss,speed_ms,0,blend_radius_m)
    |   speed_ms = 0.035
    |   movel([0.171912, -1.367931, -2.579550, -0.764907, 1.570796, 1.742708],accel_mss,speed_ms,0,blend_radius_m)
    |   movel([0.168786, -1.368788, -2.578960, -0.764640, 1.570796, 1.739583],accel_mss,speed_ms,0,blend_radius_m)
    |   movel([0.167425, -1.368959, -2.578842, -0.764588, 1.570796, 1.738221],accel_mss,speed_ms,0,blend_radius_m)
    |   movel([0.167255, -1.368826, -2.578934, -0.764629, 1.570796, 1.738052],accel_mss,speed_ms,0,blend_radius_m)
    |   movel([0.167375, -1.368564, -2.579114, -0.764710, 1.570796, 1.738171],accel_mss,speed_ms,0,blend_radius_m)
    |   movel([0.167815, -1.368296, -2.579299, -0.764794, 1.570796, 1.738611],accel_mss,speed_ms,0,blend_radius_m)
    |   movel([0.189361, -1.361530, -2.583925, -0.766933, 1.570796, 1.760157],accel_mss,speed_ms,0,blend_radius_m)
    |   movel([0.192313, -1.360743, -2.584460, -0.767186, 1.570796, 1.763109],accel_mss,speed_ms,0,blend_radius_m)
    |   movel([0.192737, -1.360754, -2.584452, -0.767183, 1.570796, 1.763534],accel_mss,speed_ms,0,blend_radius_m)
    |   movel([0.192862, -1.360992, -2.584291, -0.767106, 1.570796, 1.763658],accel_mss,speed_ms,0,blend_radius_m)
    |   movel([0.191428, -1.361791, -2.583748, -0.766849, 1.570796, 1.762224],accel_mss,speed_ms,0,blend_radius_m)
    |   movel([0.190579, -1.362091, -2.583545, -0.766753, 1.570796, 1.761375],accel_mss,speed_ms,0,blend_radius_m)
    |   movel([0.188019, -1.362877, -2.583010, -0.766502, 1.570796, 1.758815],accel_mss,speed_ms,0,blend_radius_m)
    |   speed_ms = 0.005
    |   movel([0.188019, -1.354086, -2.578929, -0.779374, 1.570796, 1.758815],accel_mss,speed_ms,0,blend_radius_m)
    |   speed_ms = 0.040
    |   movel([0.192708, -1.350089, -2.581604, -0.780696, 1.570796, 1.763505],accel_mss,speed_ms,0,blend_radius_m)
    |   speed_ms = 0.005
    |   movel([0.192708, -1.358906, -2.585702, -0.767780, 1.570796, 1.763505],accel_mss,speed_ms,0,blend_radius_m)
    |   speed_ms = 0.035
    |   movel([0.192968, -1.358766, -2.585797, -0.767826, 1.570796, 1.763764],accel_mss,speed_ms,0,blend_radius_m)
    |   movel([0.193123, -1.358527, -2.585958, -0.767904, 1.570796, 1.763920],accel_mss,speed_ms,0,blend_radius_m)
    |   movel([0.193962, -1.355315, -2.588119, -0.768955, 1.570796, 1.764759],accel_mss,speed_ms,0,blend_radius_m)
    |   movel([0.197033, -1.341780, -2.597064, -0.773545, 1.570796, 1.767830],accel_mss,speed_ms,0,blend_radius_m)
    |   movel([0.200872, -1.324330, -2.608228, -0.779831, 1.570796, 1.771668],accel_mss,speed_ms,0,blend_radius_m)
    |   movel([0.188606, -1.327232, -2.606399, -0.778757, 1.570796, 1.759402],accel_mss,speed_ms,0,blend_radius_m)
    |   movel([0.176356, -1.330244, -2.604490, -0.777654, 1.570796, 1.747152],accel_mss,speed_ms,0,blend_radius_m)
    |   movel([0.169216, -1.365805, -2.581010, -0.765574, 1.570796, 1.740012],accel_mss,speed_ms,0,blend_radius_m)
    |   movel([0.170610, -1.365485, -2.581229, -0.765675, 1.570796, 1.741407],accel_mss,speed_ms,0,blend_radius_m)
    |   movel([0.174533, -1.364346, -2.582008, -0.766035, 1.570796, 1.745329],accel_mss,speed_ms,0,blend_radius_m)
    |   movel([0.178080, -1.363276, -2.582738, -0.766375, 1.570796, 1.748877],accel_mss,speed_ms,0,blend_radius_m)
    |   movel([0.192708, -1.358906, -2.585702, -0.767780, 1.570796, 1.763505],accel_mss,speed_ms,0,blend_radius_m)
    |   movel([0.192968, -1.358766, -2.585797, -0.767826, 1.570796, 1.763764],accel_mss,speed_ms,0,blend_radius_m)
    |   movel([0.193123, -1.358527, -2.585958, -0.767904, 1.570796, 1.763920],accel_mss,speed_ms,0,blend_radius_m)
    |   movel([0.193605, -1.356686, -2.587198, -0.768505, 1.570796, 1.764402],accel_mss,speed_ms,0,blend_radius_m)
    |   speed_ms = 0.005
    |   movel([0.193605, -1.347854, -2.583091, -0.781445, 1.570796, 1.764402],accel_mss,speed_ms,0,blend_radius_m)
    |   speed_ms = 0.040
    |   movel([0.160550, -1.338801, -2.589040, -0.784548, 1.570796, 1.731347],accel_mss,speed_ms,0,blend_radius_m)
    |   speed_ms = 0.005
    |   movel([0.160550, -1.347692, -2.593188, -0.771509, 1.570796, 1.731347],accel_mss,speed_ms,0,blend_radius_m)
    |   speed_ms = 0.035
    |   movel([0.160879, -1.348502, -2.592653, -0.771234, 1.570796, 1.731676],accel_mss,speed_ms,0,blend_radius_m)
    |   movel([0.160955, -1.349444, -2.592030, -0.770915, 1.570796, 1.731751],accel_mss,speed_ms,0,blend_radius_m)
    |   movel([0.160781, -1.350501, -2.591330, -0.770559, 1.570796, 1.731577],accel_mss,speed_ms,0,blend_radius_m)
    |   movel([0.160375, -1.351592, -2.590605, -0.770192, 1.570796, 1.731171],accel_mss,speed_ms,0,blend_radius_m)
    |   movel([0.159760, -1.352660, -2.589893, -0.769836, 1.570796, 1.730557],accel_mss,speed_ms,0,blend_radius_m)
    |   movel([0.158955, -1.353676, -2.589215, -0.769497, 1.570796, 1.729752],accel_mss,speed_ms,0,blend_radius_m)
    |   movel([0.158031, -1.354543, -2.588636, -0.769210, 1.570796, 1.728828],accel_mss,speed_ms,0,blend_radius_m)
    |   movel([0.156989, -1.355259, -2.588156, -0.768974, 1.570796, 1.727785],accel_mss,speed_ms,0,blend_radius_m)
    |   movel([0.156141, -1.355820, -2.587780, -0.768789, 1.570796, 1.726937],accel_mss,speed_ms,0,blend_radius_m)
    |   movel([0.155657, -1.356332, -2.587436, -0.768621, 1.570796, 1.726453],accel_mss,speed_ms,0,blend_radius_m)
    |   movel([0.155358, -1.356992, -2.586993, -0.768404, 1.570796, 1.726154],accel_mss,speed_ms,0,blend_radius_m)
    |   movel([0.155108, -1.358136, -2.586222, -0.768031, 1.570796, 1.725904],accel_mss,speed_ms,0,blend_radius_m)
    |   movel([0.154881, -1.359235, -2.585480, -0.767674, 1.570796, 1.725678],accel_mss,speed_ms,0,blend_radius_m)
    |   movel([0.154637, -1.359810, -2.585092, -0.767488, 1.570796, 1.725433],accel_mss,speed_ms,0,blend_radius_m)
    |   movel([0.154285, -1.360149, -2.584862, -0.767378, 1.570796, 1.725082],accel_mss,speed_ms,0,blend_radius_m)
    |   movel([0.153742, -1.360373, -2.584710, -0.767306, 1.570796, 1.724538],accel_mss,speed_ms,0,blend_radius_m)
    |   movel([0.153233, -1.360404, -2.584689, -0.767296, 1.570796, 1.724029],accel_mss,speed_ms,0,blend_radius_m)
    |   movel([0.152972, -1.360208, -2.584822, -0.767359, 1.570796, 1.723768],accel_mss,speed_ms,0,blend_radius_m)
    |   movel([0.152919, -1.359698, -2.585167, -0.767524, 1.570796, 1.723715],accel_mss,speed_ms,0,blend_radius_m)
    |   movel([0.153078, -1.358581, -2.585922, -0.767886, 1.570796, 1.723874],accel_mss,speed_ms,0,blend_radius_m)
    |   movel([0.153218, -1.357576, -2.586600, -0.768214, 1.570796, 1.724014],accel_mss,speed_ms,0,blend_radius_m)
    |   movel([0.153183, -1.357016, -2.586977, -0.768397, 1.570796, 1.723979],accel_mss,speed_ms,0,blend_radius_m)
    |   movel([0.152988, -1.356758, -2.587150, -0.768481, 1.570796, 1.723784],accel_mss,speed_ms,0,blend_radius_m)
    |   movel([0.152628, -1.356732, -2.587168, -0.768490, 1.570796, 1.723424],accel_mss,speed_ms,0,blend_radius_m)
    |   movel([0.152234, -1.356749, -2.587156, -0.768484, 1.570796, 1.723030],accel_mss,speed_ms,0,blend_radius_m)
    |   movel([0.151686, -1.356590, -2.587263, -0.768536, 1.570796, 1.722482],accel_mss,speed_ms,0,blend_radius_m)
    |   movel([0.151100, -1.356323, -2.587442, -0.768624, 1.570796, 1.721896],accel_mss,speed_ms,0,blend_radius_m)
    |   movel([0.149920, -1.355380, -2.588075, -0.768934, 1.570796, 1.720717],accel_mss,speed_ms,0,blend_radius_m)
    |   movel([0.149599, -1.354787, -2.588472, -0.769129, 1.570796, 1.720395],accel_mss,speed_ms,0,blend_radius_m)
    |   movel([0.149517, -1.354025, -2.588982, -0.769382, 1.570796, 1.720313],accel_mss,speed_ms,0,blend_radius_m)
    |   movel([0.149643, -1.352885, -2.589743, -0.769760, 1.570796, 1.720439],accel_mss,speed_ms,0,blend_radius_m)
    |   movel([0.149909, -1.351709, -2.590527, -0.770153, 1.570796, 1.720705],accel_mss,speed_ms,0,blend_radius_m)
    |   movel([0.150269, -1.350831, -2.591110, -0.770448, 1.570796, 1.721066],accel_mss,speed_ms,0,blend_radius_m)
    |   movel([0.150833, -1.350012, -2.591654, -0.770723, 1.570796, 1.721629],accel_mss,speed_ms,0,blend_radius_m)
    |   movel([0.151741, -1.349028, -2.592306, -0.771056, 1.570796, 1.722537],accel_mss,speed_ms,0,blend_radius_m)
    |   movel([0.153208, -1.347747, -2.593152, -0.771490, 1.570796, 1.724004],accel_mss,speed_ms,0,blend_radius_m)
    |   movel([0.153869, -1.347283, -2.593458, -0.771648, 1.570796, 1.724665],accel_mss,speed_ms,0,blend_radius_m)
    |   movel([0.154297, -1.347094, -2.593582, -0.771713, 1.570796, 1.725093],accel_mss,speed_ms,0,blend_radius_m)
    |   movel([0.154704, -1.346875, -2.593727, -0.771787, 1.570796, 1.725500],accel_mss,speed_ms,0,blend_radius_m)
    |   movel([0.155013, -1.346488, -2.593982, -0.771920, 1.570796, 1.725810],accel_mss,speed_ms,0,blend_radius_m)
    |   movel([0.155259, -1.345848, -2.594402, -0.772139, 1.570796, 1.726055],accel_mss,speed_ms,0,blend_radius_m)
    |   movel([0.155476, -1.344805, -2.595087, -0.772497, 1.570796, 1.726272],accel_mss,speed_ms,0,blend_radius_m)
    |   movel([0.155689, -1.343786, -2.595755, -0.772849, 1.570796, 1.726485],accel_mss,speed_ms,0,blend_radius_m)
    |   movel([0.155934, -1.343135, -2.596180, -0.773074, 1.570796, 1.726731],accel_mss,speed_ms,0,blend_radius_m)
    |   movel([0.156238, -1.342736, -2.596441, -0.773212, 1.570796, 1.727034],accel_mss,speed_ms,0,blend_radius_m)
    |   movel([0.156621, -1.342517, -2.596584, -0.773288, 1.570796, 1.727418],accel_mss,speed_ms,0,blend_radius_m)
    |   movel([0.156957, -1.342544, -2.596566, -0.773279, 1.570796, 1.727753],accel_mss,speed_ms,0,blend_radius_m)
    |   movel([0.157146, -1.342795, -2.596402, -0.773192, 1.570796, 1.727942],accel_mss,speed_ms,0,blend_radius_m)
    |   movel([0.157187, -1.343319, -2.596060, -0.773010, 1.570796, 1.727983],accel_mss,speed_ms,0,blend_radius_m)
    |   movel([0.157070, -1.344191, -2.595490, -0.772709, 1.570796, 1.727867],accel_mss,speed_ms,0,blend_radius_m)
    |   movel([0.156944, -1.345243, -2.594799, -0.772346, 1.570796, 1.727740],accel_mss,speed_ms,0,blend_radius_m)
    |   movel([0.157062, -1.345795, -2.594437, -0.772157, 1.570796, 1.727858],accel_mss,speed_ms,0,blend_radius_m)
    |   movel([0.157463, -1.346123, -2.594222, -0.772045, 1.570796, 1.728260],accel_mss,speed_ms,0,blend_radius_m)
    |   movel([0.158990, -1.346558, -2.593936, -0.771896, 1.570796, 1.729786],accel_mss,speed_ms,0,blend_radius_m)
    |   movel([0.159643, -1.346882, -2.593722, -0.771785, 1.570796, 1.730439],accel_mss,speed_ms,0,blend_radius_m)
    |   movel([0.160550, -1.347692, -2.593188, -0.771509, 1.570796, 1.731347],accel_mss,speed_ms,0,blend_radius_m)
    |   movel([0.160879, -1.348502, -2.592653, -0.771234, 1.570796, 1.731676],accel_mss,speed_ms,0,blend_radius_m)
    |   movel([0.160955, -1.349444, -2.592030, -0.770915, 1.570796, 1.731751],accel_mss,speed_ms,0,blend_radius_m)
    |   movel([0.160913, -1.349691, -2.591867, -0.770832, 1.570796, 1.731709],accel_mss,speed_ms,0,blend_radius_m)
    |   speed_ms = 0.005
    |   movel([0.160913, -1.340812, -2.587728, -0.783849, 1.570796, 1.731709],accel_mss,speed_ms,0,blend_radius_m)
    |   speed_ms = 0.040
    |   movel([0.142079, -1.343658, -2.585862, -0.782869, 1.570796, 1.712875],accel_mss,speed_ms,0,blend_radius_m)
    |   speed_ms = 0.005
    |   movel([0.142079, -1.352517, -2.589988, -0.769883, 1.570796, 1.712875],accel_mss,speed_ms,0,blend_radius_m)
    |   speed_ms = 0.035
    |   movel([0.142414, -1.353633, -2.589244, -0.769512, 1.570796, 1.713211],accel_mss,speed_ms,0,blend_radius_m)
    |   movel([0.142434, -1.354438, -2.588706, -0.769245, 1.570796, 1.713231],accel_mss,speed_ms,0,blend_radius_m)
    |   movel([0.142151, -1.355327, -2.588110, -0.768951, 1.570796, 1.712947],accel_mss,speed_ms,0,blend_radius_m)
    |   movel([0.141422, -1.356731, -2.587168, -0.768490, 1.570796, 1.712218],accel_mss,speed_ms,0,blend_radius_m)
    |   movel([0.140871, -1.357564, -2.586608, -0.768217, 1.570796, 1.711667],accel_mss,speed_ms,0,blend_radius_m)
    |   movel([0.140186, -1.358355, -2.586075, -0.767960, 1.570796, 1.710982],accel_mss,speed_ms,0,blend_radius_m)
    |   movel([0.139387, -1.359081, -2.585585, -0.767724, 1.570796, 1.710184],accel_mss,speed_ms,0,blend_radius_m)
    |   movel([0.138495, -1.359722, -2.585151, -0.767516, 1.570796, 1.709291],accel_mss,speed_ms,0,blend_radius_m)
    |   movel([0.137408, -1.360472, -2.584643, -0.767274, 1.570796, 1.708205],accel_mss,speed_ms,0,blend_radius_m)
    |   movel([0.136841, -1.361036, -2.584261, -0.767092, 1.570796, 1.707637],accel_mss,speed_ms,0,blend_radius_m)
    |   movel([0.136514, -1.361674, -2.583828, -0.766887, 1.570796, 1.707311],accel_mss,speed_ms,0,blend_radius_m)
    |   movel([0.136296, -1.362671, -2.583150, -0.766568, 1.570796, 1.707092],accel_mss,speed_ms,0,blend_radius_m)
    |   movel([0.136131, -1.363484, -2.582596, -0.766309, 1.570796, 1.706927],accel_mss,speed_ms,0,blend_radius_m)
    |   movel([0.135914, -1.364033, -2.582222, -0.766134, 1.570796, 1.706710],accel_mss,speed_ms,0,blend_radius_m)
    |   movel([0.135631, -1.364383, -2.581983, -0.766023, 1.570796, 1.706427],accel_mss,speed_ms,0,blend_radius_m)
    |   movel([0.135269, -1.364580, -2.581848, -0.765961, 1.570796, 1.706065],accel_mss,speed_ms,0,blend_radius_m)
    |   movel([0.134940, -1.364561, -2.581861, -0.765967, 1.570796, 1.705737],accel_mss,speed_ms,0,blend_radius_m)
    |   movel([0.134746, -1.364334, -2.582016, -0.766039, 1.570796, 1.705543],accel_mss,speed_ms,0,blend_radius_m)
    |   movel([0.134688, -1.363856, -2.582342, -0.766190, 1.570796, 1.705484],accel_mss,speed_ms,0,blend_radius_m)
    |   movel([0.134770, -1.363066, -2.582881, -0.766442, 1.570796, 1.705567],accel_mss,speed_ms,0,blend_radius_m)
    |   movel([0.134855, -1.362104, -2.583536, -0.766749, 1.570796, 1.705651],accel_mss,speed_ms,0,blend_radius_m)
    |   movel([0.134706, -1.361589, -2.583885, -0.766914, 1.570796, 1.705503],accel_mss,speed_ms,0,blend_radius_m)
    |   movel([0.134273, -1.361285, -2.584092, -0.767012, 1.570796, 1.705070],accel_mss,speed_ms,0,blend_radius_m)
    |   movel([0.133339, -1.361060, -2.584245, -0.767084, 1.570796, 1.704135],accel_mss,speed_ms,0,blend_radius_m)
    |   movel([0.132197, -1.360656, -2.584518, -0.767214, 1.570796, 1.702994],accel_mss,speed_ms,0,blend_radius_m)
    |   movel([0.131369, -1.359907, -2.585026, -0.767456, 1.570796, 1.702165],accel_mss,speed_ms,0,blend_radius_m)
    |   movel([0.130923, -1.358869, -2.585728, -0.767793, 1.570796, 1.701719],accel_mss,speed_ms,0,blend_radius_m)
    |   movel([0.130893, -1.357616, -2.586572, -0.768200, 1.570796, 1.701690],accel_mss,speed_ms,0,blend_radius_m)
    |   movel([0.131287, -1.356234, -2.587502, -0.768653, 1.570796, 1.702083],accel_mss,speed_ms,0,blend_radius_m)
    |   movel([0.132070, -1.354842, -2.588436, -0.769112, 1.570796, 1.702866],accel_mss,speed_ms,0,blend_radius_m)
    |   movel([0.133193, -1.353526, -2.589315, -0.769547, 1.570796, 1.703990],accel_mss,speed_ms,0,blend_radius_m)
    |   movel([0.134560, -1.352399, -2.590067, -0.769923, 1.570796, 1.705357],accel_mss,speed_ms,0,blend_radius_m)
    |   movel([0.135719, -1.351547, -2.590634, -0.770207, 1.570796, 1.706516],accel_mss,speed_ms,0,blend_radius_m)
    |   movel([0.136327, -1.350927, -2.591047, -0.770416, 1.570796, 1.707123],accel_mss,speed_ms,0,blend_radius_m)
    |   movel([0.136673, -1.350258, -2.591491, -0.770640, 1.570796, 1.707469],accel_mss,speed_ms,0,blend_radius_m)
    |   movel([0.136900, -1.349258, -2.592153, -0.770978, 1.570796, 1.707696],accel_mss,speed_ms,0,blend_radius_m)
    |   movel([0.137068, -1.348445, -2.592691, -0.771253, 1.570796, 1.707865],accel_mss,speed_ms,0,blend_radius_m)
    |   movel([0.137289, -1.347889, -2.593058, -0.771442, 1.570796, 1.708085],accel_mss,speed_ms,0,blend_radius_m)
    |   movel([0.137578, -1.347533, -2.593293, -0.771563, 1.570796, 1.708374],accel_mss,speed_ms,0,blend_radius_m)
    |   movel([0.137947, -1.347329, -2.593427, -0.771632, 1.570796, 1.708743],accel_mss,speed_ms,0,blend_radius_m)
    |   movel([0.138282, -1.347347, -2.593416, -0.771626, 1.570796, 1.709078],accel_mss,speed_ms,0,blend_radius_m)
    |   movel([0.138479, -1.347579, -2.593262, -0.771547, 1.570796, 1.709275],accel_mss,speed_ms,0,blend_radius_m)
    |   movel([0.138536, -1.348069, -2.592939, -0.771381, 1.570796, 1.709332],accel_mss,speed_ms,0,blend_radius_m)
    |   movel([0.138449, -1.348878, -2.592405, -0.771106, 1.570796, 1.709245],accel_mss,speed_ms,0,blend_radius_m)
    |   movel([0.138359, -1.349860, -2.591754, -0.770774, 1.570796, 1.709155],accel_mss,speed_ms,0,blend_radius_m)
    |   movel([0.138507, -1.350384, -2.591407, -0.770598, 1.570796, 1.709303],accel_mss,speed_ms,0,blend_radius_m)
    |   movel([0.138943, -1.350693, -2.591202, -0.770494, 1.570796, 1.709739],accel_mss,speed_ms,0,blend_radius_m)
    |   movel([0.139883, -1.350924, -2.591049, -0.770417, 1.570796, 1.710679],accel_mss,speed_ms,0,blend_radius_m)
    |   movel([0.140618, -1.351134, -2.590909, -0.770346, 1.570796, 1.711414],accel_mss,speed_ms,0,blend_radius_m)
    |   movel([0.141262, -1.351491, -2.590672, -0.770226, 1.570796, 1.712058],accel_mss,speed_ms,0,blend_radius_m)
    |   movel([0.141761, -1.351964, -2.590357, -0.770068, 1.570796, 1.712557],accel_mss,speed_ms,0,blend_radius_m)
    |   movel([0.142079, -1.352517, -2.589988, -0.769883, 1.570796, 1.712875],accel_mss,speed_ms,0,blend_radius_m)
    |   movel([0.142414, -1.353633, -2.589244, -0.769512, 1.570796, 1.713211],accel_mss,speed_ms,0,blend_radius_m)
    |   movel([0.142434, -1.354438, -2.588706, -0.769245, 1.570796, 1.713231],accel_mss,speed_ms,0,blend_radius_m)
    |   speed_ms = 0.005
    |   movel([0.142434, -1.345591, -2.584588, -0.782210, 1.570796, 1.713231],accel_mss,speed_ms,0,blend_radius_m)
    |   speed_ms = 0.040
    |   movel([0.114436, -1.333669, -2.592364, -0.786357, 1.570796, 1.685232],accel_mss,speed_ms,0,blend_radius_m)
    |   speed_ms = 0.005
    |   movel([0.114436, -1.342593, -2.596534, -0.773262, 1.570796, 1.685232],accel_mss,speed_ms,0,blend_radius_m)
    |   speed_ms = 0.035
    |   movel([0.113833, -1.343560, -2.595902, -0.772927, 1.570796, 1.684629],accel_mss,speed_ms,0,blend_radius_m)
    |   movel([0.113126, -1.344496, -2.595289, -0.772603, 1.570796, 1.683923],accel_mss,speed_ms,0,blend_radius_m)
    |   movel([0.111407, -1.346304, -2.594103, -0.771983, 1.570796, 1.682203],accel_mss,speed_ms,0,blend_radius_m)
    |   movel([0.110416, -1.347147, -2.593547, -0.771694, 1.570796, 1.681212],accel_mss,speed_ms,0,blend_radius_m)
    |   movel([0.108276, -1.348623, -2.592573, -0.771193, 1.570796, 1.679072],accel_mss,speed_ms,0,blend_radius_m)
    |   movel([0.107148, -1.349245, -2.592162, -0.770982, 1.570796, 1.677945],accel_mss,speed_ms,0,blend_radius_m)
    |   movel([0.104917, -1.350171, -2.591549, -0.770670, 1.570796, 1.675714],accel_mss,speed_ms,0,blend_radius_m)
    |   movel([0.103808, -1.350478, -2.591344, -0.770566, 1.570796, 1.674604],accel_mss,speed_ms,0,blend_radius_m)
    |   movel([0.101648, -1.350769, -2.591151, -0.770468, 1.570796, 1.672444],accel_mss,speed_ms,0,blend_radius_m)
    |   movel([0.100622, -1.350750, -2.591164, -0.770475, 1.570796, 1.671418],accel_mss,speed_ms,0,blend_radius_m)
    |   movel([0.098747, -1.350392, -2.591402, -0.770595, 1.570796, 1.669544],accel_mss,speed_ms,0,blend_radius_m)
    |   movel([0.097947, -1.350065, -2.591619, -0.770705, 1.570796, 1.668744],accel_mss,speed_ms,0,blend_radius_m)
    |   movel([0.096622, -1.349105, -2.592254, -0.771029, 1.570796, 1.667419],accel_mss,speed_ms,0,blend_radius_m)
    |   movel([0.096111, -1.348485, -2.592664, -0.771239, 1.570796, 1.666907],accel_mss,speed_ms,0,blend_radius_m)
    |   movel([0.095740, -1.347814, -2.593108, -0.771467, 1.570796, 1.666536],accel_mss,speed_ms,0,blend_radius_m)
    |   movel([0.095501, -1.347061, -2.593604, -0.771724, 1.570796, 1.666297],accel_mss,speed_ms,0,blend_radius_m)
    |   movel([0.095395, -1.346236, -2.594147, -0.772006, 1.570796, 1.666191],accel_mss,speed_ms,0,blend_radius_m)
    |   movel([0.095426, -1.345354, -2.594727, -0.772308, 1.570796, 1.666222],accel_mss,speed_ms,0,blend_radius_m)
    |   movel([0.095866, -1.343230, -2.596118, -0.773041, 1.570796, 1.666663],accel_mss,speed_ms,0,blend_radius_m)
    |   movel([0.096222, -1.342257, -2.596753, -0.773379, 1.570796, 1.667018],accel_mss,speed_ms,0,blend_radius_m)
    |   movel([0.096705, -1.341277, -2.597392, -0.773720, 1.570796, 1.667501],accel_mss,speed_ms,0,blend_radius_m)
    |   movel([0.097043, -1.340834, -2.597680, -0.773875, 1.570796, 1.667839],accel_mss,speed_ms,0,blend_radius_m)
    |   movel([0.097498, -1.340479, -2.597911, -0.773999, 1.570796, 1.668295],accel_mss,speed_ms,0,blend_radius_m)
    |   movel([0.097874, -1.340383, -2.597973, -0.774033, 1.570796, 1.668670],accel_mss,speed_ms,0,blend_radius_m)
    |   movel([0.098443, -1.340848, -2.597671, -0.773870, 1.570796, 1.669239],accel_mss,speed_ms,0,blend_radius_m)
    |   movel([0.098748, -1.340902, -2.597636, -0.773851, 1.570796, 1.669544],accel_mss,speed_ms,0,blend_radius_m)
    |   movel([0.099687, -1.340837, -2.597678, -0.773874, 1.570796, 1.670484],accel_mss,speed_ms,0,blend_radius_m)
    |   movel([0.100230, -1.340920, -2.597624, -0.773845, 1.570796, 1.671026],accel_mss,speed_ms,0,blend_radius_m)
    |   movel([0.101769, -1.341496, -2.597249, -0.773644, 1.570796, 1.672565],accel_mss,speed_ms,0,blend_radius_m)
    |   movel([0.103166, -1.342298, -2.596727, -0.773364, 1.570796, 1.673962],accel_mss,speed_ms,0,blend_radius_m)
    |   movel([0.103885, -1.343124, -2.596187, -0.773078, 1.570796, 1.674681],accel_mss,speed_ms,0,blend_radius_m)
    |   movel([0.104469, -1.343720, -2.595797, -0.772871, 1.570796, 1.675266],accel_mss,speed_ms,0,blend_radius_m)
    |   movel([0.104853, -1.343839, -2.595720, -0.772830, 1.570796, 1.675649],accel_mss,speed_ms,0,blend_radius_m)
    |   movel([0.105311, -1.343824, -2.595730, -0.772836, 1.570796, 1.676107],accel_mss,speed_ms,0,blend_radius_m)
    |   movel([0.105774, -1.343681, -2.595823, -0.772885, 1.570796, 1.676570],accel_mss,speed_ms,0,blend_radius_m)
    |   movel([0.106227, -1.343413, -2.595998, -0.772977, 1.570796, 1.677023],accel_mss,speed_ms,0,blend_radius_m)
    |   movel([0.107036, -1.342586, -2.596539, -0.773264, 1.570796, 1.677832],accel_mss,speed_ms,0,blend_radius_m)
    |   movel([0.107279, -1.342147, -2.596825, -0.773417, 1.570796, 1.678075],accel_mss,speed_ms,0,blend_radius_m)
    |   movel([0.107400, -1.341711, -2.597109, -0.773569, 1.570796, 1.678197],accel_mss,speed_ms,0,blend_radius_m)
    |   movel([0.107388, -1.341320, -2.597364, -0.773705, 1.570796, 1.678184],accel_mss,speed_ms,0,blend_radius_m)
    |   movel([0.106943, -1.340726, -2.597750, -0.773913, 1.570796, 1.677739],accel_mss,speed_ms,0,blend_radius_m)
    |   movel([0.106546, -1.340559, -2.597859, -0.773971, 1.570796, 1.677343],accel_mss,speed_ms,0,blend_radius_m)
    |   movel([0.104127, -1.340352, -2.597994, -0.774044, 1.570796, 1.674923],accel_mss,speed_ms,0,blend_radius_m)
    |   movel([0.102587, -1.339822, -2.598337, -0.774229, 1.570796, 1.673384],accel_mss,speed_ms,0,blend_radius_m)
    |   movel([0.101253, -1.339138, -2.598781, -0.774470, 1.570796, 1.672050],accel_mss,speed_ms,0,blend_radius_m)
    |   movel([0.101043, -1.338896, -2.598938, -0.774555, 1.570796, 1.671839],accel_mss,speed_ms,0,blend_radius_m)
    |   movel([0.100948, -1.338356, -2.599288, -0.774746, 1.570796, 1.671745],accel_mss,speed_ms,0,blend_radius_m)
    |   movel([0.100740, -1.338203, -2.599387, -0.774800, 1.570796, 1.671536],accel_mss,speed_ms,0,blend_radius_m)
    |   movel([0.099656, -1.338024, -2.599502, -0.774863, 1.570796, 1.670452],accel_mss,speed_ms,0,blend_radius_m)
    |   movel([0.100127, -1.337368, -2.599926, -0.775095, 1.570796, 1.670924],accel_mss,speed_ms,0,blend_radius_m)
    |   movel([0.101463, -1.336390, -2.600556, -0.775442, 1.570796, 1.672259],accel_mss,speed_ms,0,blend_radius_m)
    |   movel([0.102861, -1.335461, -2.601155, -0.775773, 1.570796, 1.673658],accel_mss,speed_ms,0,blend_radius_m)
